FUNCTION_BLOCK "TYPIC_C401_IF_RSS"   // FB106, FBD
TITLE = TYPIC_C401_IF_RSS: RSS-bord
{ S7_Optimized_Access := 'TRUE' }
AUTHOR : OCOTECH
FAMILY : Typical
NAME : C401.701
// Logisch Object Besturing: C401.701
// 
// De interne functie RSSobord verzorgt de bewaking van een RSSobord en stuurt de informatie door naar de subfunctie.
// stored: MemoryReserve 10, SetENOAutomatically false
   VAR_INPUT
      EXT_AUT { ExternalAccessible := 'False'; ExternalVisible := 'False'; ExternalWritable := 'False'} : Bool;   // Externe (hoofd) beveiliging (1 = OK)
      EXT_HW { ExternalAccessible := 'False'; ExternalVisible := 'False'; ExternalWritable := 'False'} : Bool;   // Sturings hardware (PLC) bewaking (1 = OK)
      IN_STO_NOK { ExternalAccessible := 'False'; ExternalVisible := 'False'; ExternalWritable := 'False'} : Bool;   // Storing aanwezig die niet observeerbaar tot gevolg heeft
      IN_STO_OK { ExternalAccessible := 'False'; ExternalVisible := 'False'; ExternalWritable := 'False'} : Bool;   // Storing aanwezig die observeerbaarheid niet beinvloed
      IN_LUS_STO { ExternalAccessible := 'False'; ExternalVisible := 'False'; ExternalWritable := 'False'} : Bool;   // Storing van het luspaar
      IN_STS { ExternalAccessible := 'False'; ExternalVisible := 'False'; ExternalWritable := 'False'} : String[8];   // Naam van de getoonde beeldstand (bitmap) op het bord
      IN_PRTG_STO { ExternalAccessible := 'False'; ExternalVisible := 'False'; ExternalWritable := 'False'} : Bool;   // Storingsmelding RSS-bord vanuit PRTG
      IN_AUT_C401 { ExternalAccessible := 'False'; ExternalVisible := 'False'; ExternalWritable := 'False'} : Bool;   // Beveiligingen: serie geschakelde terugmelding (1 = OK)
   END_VAR
   VAR_OUTPUT
      VAR_IF_RSS { ExternalAccessible := 'False'; ExternalVisible := 'False'; ExternalWritable := 'False'} : "C401_VAR_IF_RSS_TYPIC";   // Struct met alle variabelen naar bovenliggende functies
   END_VAR
   VAR
      STO { ExternalWritable := 'False'} : Struct   // Storingen
         A001 { ExternalAccessible := 'False'; ExternalVisible := 'False'} : Bool;   // Beveiliging aangesproken
         A002 { ExternalAccessible := 'False'; ExternalVisible := 'False'} : Bool;   // Storing luspaar
         A003 { ExternalAccessible := 'False'; ExternalVisible := 'False'} : Bool;   // Storing RSS-bord gedetecteerd door PRTG
         A004 { ExternalAccessible := 'False'; ExternalVisible := 'False'} : Bool;   // Storing RSS-bord
         A005 { ExternalAccessible := 'False'; ExternalVisible := 'False'} : Bool;   // Algemene storing RSS-bord
      END_STRUCT;
      VAR { ExternalWritable := 'False'} : Struct   // Variabelen
         STS { ExternalAccessible := 'False'; ExternalVisible := 'False'} : String[8];   // Naam van de getoonde beeldstand (bitmap) op het bord
         EXT_AUT { ExternalAccessible := 'False'; ExternalVisible := 'False'} : Bool;   // Externe (hoofd) beveiliging aangesproken
         EXT_HW { ExternalAccessible := 'False'; ExternalVisible := 'False'} : Bool;   // Sturings hardware (PLC) in storing
      END_STRUCT;
   END_VAR
BEGIN

REGION Network 1: START
END_REGION

REGION Network 2: +++ Storingen +++
   // Verzamelen storingsmeldingen.
END_REGION

REGION Network 3: Storing A001: Beveiliging aangesproken
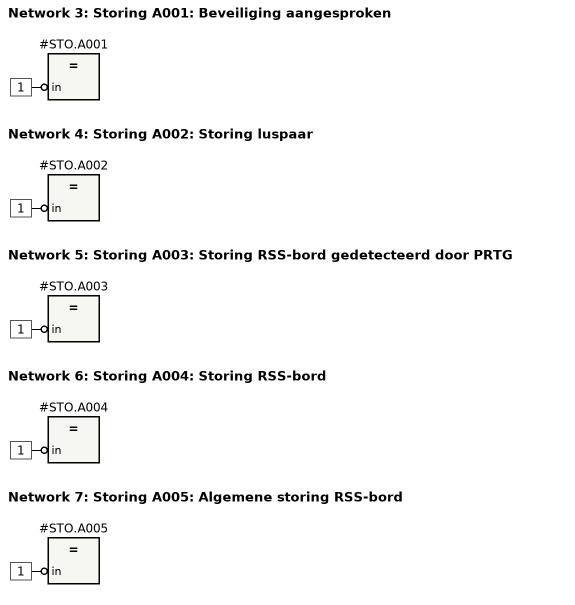
   #STO.A001 := NOT 1;
END_REGION

REGION Network 4: Storing A002: Storing luspaar
   #STO.A002 := NOT 1;
END_REGION

REGION Network 5: Storing A003: Storing RSS-bord gedetecteerd door PRTG
   #STO.A003 := NOT 1;
END_REGION

REGION Network 6: Storing A004: Storing RSS-bord
   #STO.A004 := NOT 1;
END_REGION

REGION Network 7: Storing A005: Algemene storing RSS-bord
   #STO.A005 := NOT 1;
END_REGION

REGION Network 8: +++ Beeldstand +++
   // Doorgeven van de status van het RSS-bord naar de subfunctie.
END_REGION

REGION Network 9 (SCL): EINDE
   // Variabelen van intern scada rakvlak naar outputs copieren
   #VAR_IF_RSS.STS := #VAR.STS;
   #VAR_IF_RSS.EXT_AUT := #VAR.EXT_AUT;
   #VAR_IF_RSS.EXT_HW := #VAR.EXT_HW;
   #VAR_IF_RSS.STO := #STO;
END_REGION
END_FUNCTION_BLOCK

FUNCTION_BLOCK "TYPIC_C402_IF_M33"   // FB110, FBD
TITLE = TYPIC_C402_IF_M33: Voorwaarschuwingsbord
{ S7_Optimized_Access := 'TRUE' }
AUTHOR : OCOTECH
FAMILY : Typical
NAME : C402.703
// Logisch Object Besturing: C402.703
// 
// De interne functie M33 verzorgt de interne besturing van een M33obord.
// 
// Een M33obord is een waarschuwingsbord “verkeerslichten”. Dit bord waarschuwt het verkeer dat zij een actief verkeerslicht naderen.
// 
// Via het DVMosysteem worden de storingsmeldingen van ieder M33obord ingelezen. DVM meldt op zijn beurt storingen van iedere M33obord rechtstreeks aan 3B. De interne besturing heeft geen communicatie met DVM.
// stored: MemoryReserve 10, SetENOAutomatically false
   VAR_INPUT
      EXT_AUT { ExternalAccessible := 'False'; ExternalVisible := 'False'; ExternalWritable := 'False'} : Bool;   // Externe (hoofd) beveiliging (1 = OK)
      EXT_HW { ExternalAccessible := 'False'; ExternalVisible := 'False'; ExternalWritable := 'False'} : Bool;   // Sturings hardware (PLC) bewaking (1 = OK)
      IN_STO_NOK { ExternalAccessible := 'False'; ExternalVisible := 'False'; ExternalWritable := 'False'} : Bool;   // Storing aanwezig die niet observeerbaar tot gevolg heeft
      IN_STO_OK { ExternalAccessible := 'False'; ExternalVisible := 'False'; ExternalWritable := 'False'} : Bool;   // Storing aanwezig die observeerbaarheid niet beinvloed
      IN_PRTG_STO { ExternalAccessible := 'False'; ExternalVisible := 'False'; ExternalWritable := 'False'} : Bool;   // Storingsmelding RSS-bord vanuit PRTG
      IN_AUT_C402 { ExternalAccessible := 'False'; ExternalVisible := 'False'; ExternalWritable := 'False'} : Bool;   // Serie geschakelde beveiligingen (1 = OK)
      IN_AAN { ExternalAccessible := 'False'; ExternalVisible := 'False'; ExternalWritable := 'False'} : Bool;   // Terugmelding aansturing M33-bord (1 = AAN)
      CFG_TYD_FB { ExternalAccessible := 'False'; ExternalVisible := 'False'; ExternalWritable := 'False'} : Time;   // Vertragingstijd storing foute terugmelding
   END_VAR
   VAR_OUTPUT
      VAR_IF_M33 { ExternalAccessible := 'False'; ExternalVisible := 'False'; ExternalWritable := 'False'} : "C402_VAR_IF_M33_TYPIC";   // Struct met alle variabelen naar bovenliggende functies
      OUT_AAN { ExternalAccessible := 'False'; ExternalVisible := 'False'; ExternalWritable := 'False'} : Bool;   // Aansturing M33-bord (TRUE = Uit / FALSE = Aan)
   END_VAR
   VAR_IN_OUT
      STU_IF_M33 : "C402_STU_IF_M33_TYPIC";   // Struct met alle sturingen van de subfunctie (SF) M33 van 3B
   END_VAR
   VAR
      STO { ExternalWritable := 'False'} : Struct   // Storingen
         A001 { ExternalAccessible := 'False'; ExternalVisible := 'False'} : Bool;   // Beveiliging aangesproken
         A002 { ExternalAccessible := 'False'; ExternalVisible := 'False'} : Bool;   // Storing M33-bord gedetecteerd door PRTG
         A003 { ExternalAccessible := 'False'; ExternalVisible := 'False'} : Bool;   // Storing M33-bord
         A004 { ExternalAccessible := 'False'; ExternalVisible := 'False'} : Bool;   // Algemene storing M33-bord
         AT01 { ExternalAccessible := 'False'; ExternalVisible := 'False'} : Bool;   // Foute terugmelding: M33-bord aangestuurd, terugmelding Aan niet (of te laat) ontvangen
         AT02 { ExternalAccessible := 'False'; ExternalVisible := 'False'} : Bool;   // Foute terugmelding: M33-bord niet aangestuurd, terugmelding Aan blijft aanwezig
      END_STRUCT;
      VAR { ExternalWritable := 'False'} : Struct   // Variabelen
         STS_AAN { ExternalAccessible := 'False'; ExternalVisible := 'False'} : Bool;   // TRUE = M33-bord actueel in werking FALSE = Uit
         EXT_AUT { ExternalAccessible := 'False'; ExternalVisible := 'False'} : Bool;   // Externe (hoofd) beveiliging aangesproken
         EXT_HW { ExternalAccessible := 'False'; ExternalVisible := 'False'} : Bool;   // Sturings hardware (PLC) in storing
      END_STRUCT;
   END_VAR
BEGIN

REGION Network 1: START
END_REGION

REGION Network 2: +++ Aansturing bord +++
   // Aansturen bord en terugmeldingsbewaking (Aan / Uit).
END_REGION

REGION Network 3: +++ Storingen +++
   // Verwerken van de storingsmeldingen.
END_REGION

REGION Network 4: Storing A001: Beveiliging aangesproken
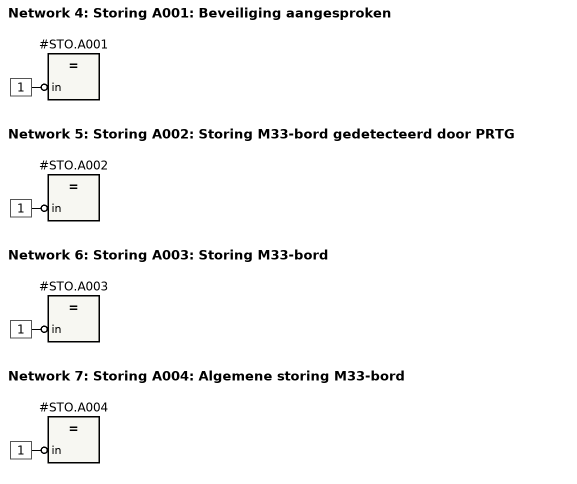
   #STO.A001 := NOT 1;
END_REGION

REGION Network 5: Storing A002: Storing M33-bord gedetecteerd door PRTG
   #STO.A002 := NOT 1;
END_REGION

REGION Network 6: Storing A003: Storing M33-bord
   #STO.A003 := NOT 1;
END_REGION

REGION Network 7: Storing A004: Algemene storing M33-bord
   #STO.A004 := NOT 1;
END_REGION

REGION Network 8 (SCL): EINDE
   // Variabelen van intern scada rakvlak naar outputs copieren
   #VAR_IF_M33.STS_AAN := #VAR.STS_AAN;
   #VAR_IF_M33.EXT_AUT := #VAR.EXT_AUT;
   #VAR_IF_M33.EXT_HW := #VAR.EXT_HW;
   #VAR_IF_M33.STO := #STO;
END_REGION
END_FUNCTION_BLOCK

FUNCTION_BLOCK "TYPIC_C402_IF_SBO1"   // FB111, FBD
TITLE = TYPIC_C402_IF_SBO: Afsluitboom
{ S7_Optimized_Access := 'TRUE' }
AUTHOR : OCOTECH
FAMILY : Typical
NAME : C402.704
// Logisch Object Besturing: C402.704
// 
// 								De interne functie afsluitboom verzorgt de interne besturing,
// 								bewaking en fysieke aansturing van een afsluitboom.
// 
// 								Het akoestisch signaal en de optische signalen behorend bij de
// 								afsluitboom, wordt eveneens via deze functie aangestuurd.
// stored: MemoryReserve 10, SetENOAutomatically false
   VAR_INPUT
      EXT_AUT { ExternalAccessible := 'False'; ExternalVisible := 'False'; ExternalWritable := 'False'} : Bool;   // Externe (hoofd) beveiliging (1 = OK)
      EXT_HW { ExternalAccessible := 'False'; ExternalVisible := 'False'; ExternalWritable := 'False'} : Bool;   // Sturings hardware (PLC) bewaking (1 = OK)
      HULP_KNIP { ExternalAccessible := 'False'; ExternalVisible := 'False'; ExternalWritable := 'False'} : Bool;   // Knippersignaal, x tijd hoog, x tijd laag
      IN_AUT { ExternalAccessible := 'False'; ExternalVisible := 'False'; ExternalWritable := 'False'} : Bool;   // Motorbeveiliging (1 = OK / 0 = storing)
      IN_OPEN { ExternalAccessible := 'False'; ExternalVisible := 'False'; ExternalWritable := 'False'} : Bool;   // Terugmelding: afsluitboom is open
      IN_TOE { ExternalAccessible := 'False'; ExternalVisible := 'False'; ExternalWritable := 'False'} : Bool;   // Terugmelding: afsluitboom is toe
      IN_STO { ExternalAccessible := 'False'; ExternalVisible := 'False'; ExternalWritable := 'False'} : Bool;   // Terugmelding: afsluitboom is buiten dienst
      IN_SCW { ExternalAccessible := 'False'; ExternalVisible := 'False'; ExternalWritable := 'False'} : Bool;   // Werkschakelaar (1 = AAN)
      IN_HND { ExternalAccessible := 'False'; ExternalVisible := 'False'; ExternalWritable := 'False'} : Bool;   // Mechanische handmatige bediening (0 = Hand)
      IN_LVE1_STO { ExternalAccessible := 'False'; ExternalVisible := 'False'; ExternalWritable := 'False'} : Bool;   // Detector lus 1 (1 = OK / 0 = storing)
      IN_LVE2_STO { ExternalAccessible := 'False'; ExternalVisible := 'False'; ExternalWritable := 'False'} : Bool;   // Detector lus 2 (1 = OK / 0 = storing)
      IN_LVE3_STO { ExternalAccessible := 'False'; ExternalVisible := 'False'; ExternalWritable := 'False'} : Bool;   // Detector lus 3 (1 = OK / 0 = storing)
      IN_LVE4_STO { ExternalAccessible := 'False'; ExternalVisible := 'False'; ExternalWritable := 'False'} : Bool;   // Detector lus 4 (1 = OK / 0 = storing)
      IN_LUS1_STS { ExternalAccessible := 'False'; ExternalVisible := 'False'; ExternalWritable := 'False'} : Bool;   // Detectie voertuig door lus 1 (1 = Geen detectie)
      IN_LUS2_STS { ExternalAccessible := 'False'; ExternalVisible := 'False'; ExternalWritable := 'False'} : Bool;   // Detectie voertuig door lus 2 (1 = Geen detectie)
      IN_LUS3_STS { ExternalAccessible := 'False'; ExternalVisible := 'False'; ExternalWritable := 'False'} : Bool;   // Detectie voertuig door lus 3 (1 = Geen detectie)
      IN_LUS4_STS { ExternalAccessible := 'False'; ExternalVisible := 'False'; ExternalWritable := 'False'} : Bool;   // Detectie voertuig door lus 4 (1 = Geen detectie)
      IN_AUT_C402 { ExternalAccessible := 'False'; ExternalVisible := 'False'; ExternalWritable := 'False'} : Bool;   // Beveiligingen: serie geschakelde terugmelding (1 = OK)
      IN_DKN_OPEN { ExternalAccessible := 'False'; ExternalVisible := 'False'; ExternalWritable := 'False'} : Bool;   // 1 = Drukknop ingedrukt, bediening openen
      IN_DKN_TOE { ExternalAccessible := 'False'; ExternalVisible := 'False'; ExternalWritable := 'False'} : Bool;   // 1 = Drukknop ingedrukt, bediening sluiten
      IN_DKN_STOP { ExternalAccessible := 'False'; ExternalVisible := 'False'; ExternalWritable := 'False'} : Bool;   // 1 = Drukknop ingedrukt, bediening stop
      CFG_TYD_STS { ExternalAccessible := 'False'; ExternalVisible := 'False'; ExternalWritable := 'False'} : Time;   // Vertragingstijd storing terugmelding stand bereikt
      CFG_ITYD_POS { ExternalAccessible := 'False'; ExternalVisible := 'False'; ExternalWritable := 'False'} : Time;   // Inschakelvertraging storing eindpositie terugmelding weggevallen
      CFG_UTYD_POS { ExternalAccessible := 'False'; ExternalVisible := 'False'; ExternalWritable := 'False'} : Time;   // Uitschakelvertraging storing eindpositie terugmelding weggevallen
      CFG_ITYD_OAS_SNEL { ExternalAccessible := 'False'; ExternalVisible := 'False'; ExternalWritable := 'False'} : Time;   // Vertragingstijd versneld sluiten afsluitboom na akoestisch en optisch signaal
      CFG_ITYD_OAS { ExternalAccessible := 'False'; ExternalVisible := 'False'; ExternalWritable := 'False'} : Time;   // Vertragingstijd sluiten/openen afsluitboom regulier na akoestisch en optisch signaal
      CFG_UTYD_OAS { ExternalAccessible := 'False'; ExternalVisible := 'False'; ExternalWritable := 'False'} : Time;   // Vertragingstijd uitschakelen akoestische en optische signalen
      CFG_UTYD_MOT { ExternalAccessible := 'False'; ExternalVisible := 'False'; ExternalWritable := 'False'} : Time;   // Vertragingstijd uitschakelen motor na bereiken eindpositie
      CFG_VGV_OPEN { ExternalAccessible := 'False'; ExternalVisible := 'False'; ExternalWritable := 'False'} : Bool;   // 1 = Slagboom moet openen bij bediening openen door hulpdiensten
   END_VAR
   VAR_OUTPUT
      VAR_IF_SBO { ExternalAccessible := 'False'; ExternalVisible := 'False'; ExternalWritable := 'False'} : "C402_VAR_IF_SBO_TYPIC";   // Struct met alle variabelen naar bovenliggende functies
      OUT_OPEN { ExternalAccessible := 'False'; ExternalVisible := 'False'; ExternalWritable := 'False'} : Bool;   // Aansturing openen
      OUT_TOE { ExternalAccessible := 'False'; ExternalVisible := 'False'; ExternalWritable := 'False'} : Bool;   // Aansturing sluiten
      OUT_AKS { ExternalAccessible := 'False'; ExternalVisible := 'False'; ExternalWritable := 'False'} : Bool;   // Aansturen akoestische signalering
      OUT_OPS { ExternalAccessible := 'False'; ExternalVisible := 'False'; ExternalWritable := 'False'} : Bool;   // Aansturen optische signalering
   END_VAR
   VAR_IN_OUT
      STU_IF_SBO : "C402_STU_IF_SBO_TYPIC";   // Struct met alle sturingen naar de functie (IF) in de interne sturing van de afsluitboom
      STU_AFS_IF_SBO : "C402_STU_AFS_IF_SBO_TYPIC";   // Struct met alle sturingen vanuit de interne functie Afsluitsysteem naar de functies (IF) van de afsluitbomen
   END_VAR
   VAR
      STO { ExternalWritable := 'False'} : Struct   // Storingen
         A001 { ExternalAccessible := 'False'; ExternalVisible := 'False'} : Bool;   // Beveiliging aangesproken
         A002 { ExternalAccessible := 'False'; ExternalVisible := 'False'} : Bool;   // Storing van de detector van lus 1
         A003 { ExternalAccessible := 'False'; ExternalVisible := 'False'} : Bool;   // Storing van de detector van lus 2
         A004 { ExternalAccessible := 'False'; ExternalVisible := 'False'} : Bool;   // Storing van de detector van lus 3
         A005 { ExternalAccessible := 'False'; ExternalVisible := 'False'} : Bool;   // Storing van de detector van lus 4
         A006 { ExternalAccessible := 'False'; ExternalVisible := 'False'} : Bool;   // Storing van de motorsturing
         A007 { ExternalAccessible := 'False'; ExternalVisible := 'False'} : Bool;   // Storing motorbeveiliging
         AT01 { ExternalAccessible := 'False'; ExternalVisible := 'False'} : Bool;   // Terugmelding Open niet tijdig bereikt
         AT02 { ExternalAccessible := 'False'; ExternalVisible := 'False'} : Bool;   // Terugmelding Dicht niet tijdig bereikt
         AT03 { ExternalAccessible := 'False'; ExternalVisible := 'False'} : Bool;   // Terugmeldingen Open en Dicht tegelijkertijd
         AT04 { ExternalAccessible := 'False'; ExternalVisible := 'False'} : Bool;   // Terugmelding Open weggevallen
         AT05 { ExternalAccessible := 'False'; ExternalVisible := 'False'} : Bool;   // Terugmelding Dicht weggevallen
         M001 { ExternalAccessible := 'False'; ExternalVisible := 'False'} : Bool;   // Werkschakelaar uitgeschakeld
         M002 { ExternalAccessible := 'False'; ExternalVisible := 'False'} : Bool;   // Mechanische handbediening uitgenomen
      END_STRUCT;
      VAR { ExternalWritable := 'False'} : Struct   // Variabelen
         CMD_AKS { ExternalAccessible := 'False'; ExternalVisible := 'False'} : Bool;   // Aansturen akoestische signalering
         CMD_OPS { ExternalAccessible := 'False'; ExternalVisible := 'False'} : Bool;   // Aansturen optische signalering
         VWA_AT04 { ExternalAccessible := 'False'; ExternalVisible := 'False'} : Bool;   // Voorwaarden voldaan voor storing AT04
         VWA_AT05 { ExternalAccessible := 'False'; ExternalVisible := 'False'} : Bool;   // Voorwaarden voldaan voor storing AT05
         MOT_STS_AAN { ExternalAccessible := 'False'; ExternalVisible := 'False'} : Bool;   // Motor afsluitboom aangestuurd
         CMD_OPEN { ExternalAccessible := 'False'; ExternalVisible := 'False'} : Bool;   // Gewenste stand afsluitboom is Open
         CMD_TOE { ExternalAccessible := 'False'; ExternalVisible := 'False'} : Bool;   // Gewenste stand afsluitboom is Toe
         CMD_STOP { ExternalAccessible := 'False'; ExternalVisible := 'False'} : Bool;   // Gewenste stand afsluitboom is Stop
         STO { ExternalAccessible := 'False'; ExternalVisible := 'False'} : Bool;   // De afsluitboom heeft een storing waardoor deze niet aangestuurd kan worden
         LOK_OPEN { ExternalAccessible := 'False'; ExternalVisible := 'False'} : Bool;   // Afsluitboom dient te openen voor hulpdiensten
         CMD_NEW { ExternalAccessible := 'False'; ExternalVisible := 'False'} : Bool;   // Nieuwe commando ontvangen vanuit 3B
         VGV_TOE { ExternalAccessible := 'False'; ExternalVisible := 'False'} : Bool;   // Vrijgave om de afsluitboom te sluiten
         CMD_TYD_OPEN { ExternalAccessible := 'False'; ExternalVisible := 'False'} : Bool;   // Gewenste stand afsluitboom is Open, tijdsvertraging OK
         CMD_TYD_TOE { ExternalAccessible := 'False'; ExternalVisible := 'False'} : Bool;   // Gewenste stand afsluitboom is Toe, tijdsvertraging OK
         STS_BEZ_OPEN { ExternalAccessible := 'False'; ExternalVisible := 'False'} : Bool;   // TRUE = Afsluitboom bezig met beweging openen
         STS_BEZ_TOE { ExternalAccessible := 'False'; ExternalVisible := 'False'} : Bool;   // TRUE = Afsluitboom bezig met beweging sluiten
         STS_OPEN { ExternalAccessible := 'False'; ExternalVisible := 'False'} : Bool;   // TRUE = Afsluitboom op stand Open
         STS_TOE { ExternalAccessible := 'False'; ExternalVisible := 'False'} : Bool;   // TRUE = Afsluitboom op stand Dicht
         STS_STOP { ExternalAccessible := 'False'; ExternalVisible := 'False'} : Bool;   // TRUE = Afsluitboom niet op een eindpositie en niet in beweging
         BMO_HAND { ExternalAccessible := 'False'; ExternalVisible := 'False'} : Bool;   // TRUE = Afsluitboom in hand geschakeld / FALSE = niet in hand
         STS_VKL_OK { ExternalAccessible := 'False'; ExternalVisible := 'False'} : Bool;   // TRUE = Verkeerslichten op Rood (voorwaarde voor sluiten)
         STS_NDS_OK { ExternalAccessible := 'False'; ExternalVisible := 'False'} : Bool;   // TRUE = Geen noodstop (voorwaarde voor beweging)
         STS_LUS_OK { ExternalAccessible := 'False'; ExternalVisible := 'False'} : Bool;   // TRUE = Detectielus(sen) OK (geen obstakel gedetecteerd voor sluiten)
         EXT_AUT { ExternalAccessible := 'False'; ExternalVisible := 'False'} : Bool;   // Externe (hoofd) beveiliging aangesproken
         EXT_HW { ExternalAccessible := 'False'; ExternalVisible := 'False'} : Bool;   // Sturings hardware (PLC) in storing
         EXT_STO { ExternalAccessible := 'False'; ExternalVisible := 'False'} : Bool;   // Externe storing aanwezig
         LUS1_STS { ExternalAccessible := 'False'; ExternalVisible := 'False'} : Bool;   // Detectie voertuig door lus 1 (1 = detectie)
         LUS2_STS { ExternalAccessible := 'False'; ExternalVisible := 'False'} : Bool;   // Detectie voertuig door lus 2 (1 = detectie)
         LUS3_STS { ExternalAccessible := 'False'; ExternalVisible := 'False'} : Bool;   // Detectie voertuig door lus 3 (1 = detectie)
         LUS4_STS { ExternalAccessible := 'False'; ExternalVisible := 'False'} : Bool;   // Detectie voertuig door lus 3 (1 = detectie)
      END_STRUCT;
   END_VAR
BEGIN

REGION Network 1: START
END_REGION

REGION Network 2: +++ Storingen en meldingen +++
   // Verwerken van de storingen en meldingen.
END_REGION

REGION Network 3: Storing A001: Beveiliging aangesproken
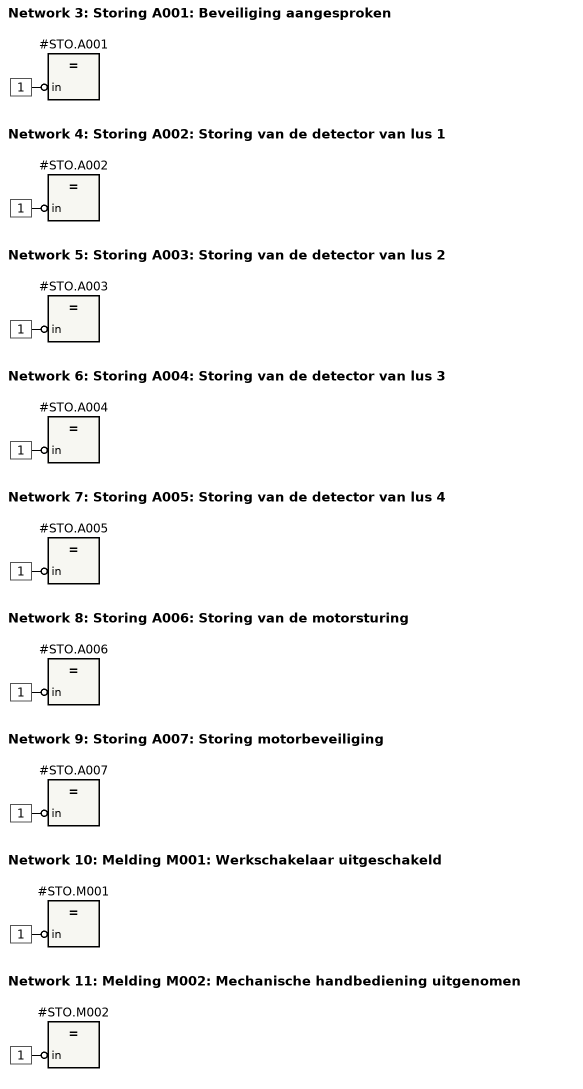
   #STO.A001 := NOT 1;
END_REGION

REGION Network 4: Storing A002: Storing van de detector van lus 1
   #STO.A002 := NOT 1;
END_REGION

REGION Network 5: Storing A003: Storing van de detector van lus 2
   #STO.A003 := NOT 1;
END_REGION

REGION Network 6: Storing A004: Storing van de detector van lus 3
   #STO.A004 := NOT 1;
END_REGION

REGION Network 7: Storing A005: Storing van de detector van lus 4
   #STO.A005 := NOT 1;
END_REGION

REGION Network 8: Storing A006: Storing van de motorsturing
   #STO.A006 := NOT 1;
END_REGION

REGION Network 9: Storing A007: Storing motorbeveiliging
   #STO.A007 := NOT 1;
END_REGION

REGION Network 10: Melding M001: Werkschakelaar uitgeschakeld
   #STO.M001 := NOT 1;
END_REGION

REGION Network 11: Melding M002: Mechanische handbediening uitgenomen
   #STO.M002 := NOT 1;
END_REGION

REGION Network 12: +++ Status detectielussen +++
   // De afsluitboom kan enkel voorwaardelijk sluiten als de
   // 										detectielussen geen metalen object detecteren en geen
   // 										storing hebben.
END_REGION

REGION Network 13: +++ Openen afsluitboom voor hulpdiensten +++
   // De afsluitboom kan door de hulpdiensten geopend worden als
   // 										op het bedieningspaneel de betreffende drukknop bediend
   // 										wordt en er vrijgave is voor bediening.
END_REGION

REGION Network 14: +++ Gewenste beweging afsluitboom +++
   // Afhankelijk van de werkingsmode, bedieningen en commandos
   // 										wordt de gewenste beweging van de afsluitboom bepaald
   // 										(openen / sluiten / stop).
END_REGION

REGION Network 15: +++ Vrijgave sluiten +++
   // Het sluiten van de afsluitboom mag enkel plaatsvinden als
   // 										er geen obstakel gedetecteerd wordt. Bij handbediening of
   // 										bij het commando onvoorwaardelijk sluiten wordt er geen
   // 										rekening gehouden met de obstakeldetectie.
END_REGION

REGION Network 16: +++ Tijdsvertraging aansturen afsluitboom +++
   // Vooraleer de afsluitboom aan te sturen, dienen de
   // 										akoestische en optische signalering aangestuurd te zijn. Pas
   // 										na een korte tijdsvertraging mag de afsluitboom in beweging
   // 										komen.
END_REGION

REGION Network 17: +++ Afsluitboomsturing +++
   // Aansturen van de afsluitboom en terugmeldingsbewaking.
END_REGION

REGION Network 18: +++ Sturing akoestische signalering +++
   // De akoestische signalering wordt aangestuurd van zodra de
   // 										afsluitboom dient te bewegen. De beweging wordt pas ingezet
   // 										nadat de akoestische signalering gedurende een bepaalde tijd
   // 										aangestuurd geweest is.
END_REGION

REGION Network 19: +++ Sturing Optische signalering +++
   // De optische signalering wordt aangestuurd van zodra de
   // 										afsluitboom dient te bewegen en blijft aangestuurd tot de
   // 										afsluitboom zich opnieuw in de open positie bevindt.
END_REGION

REGION Network 20 (SCL): EINDE
   // Variabelen van intern scada rakvlak naar outputs copieren
   #VAR_IF_SBO.STS_BEZ_OPEN := #VAR.STS_BEZ_OPEN;
   #VAR_IF_SBO.STS_BEZ_TOE := #VAR.STS_BEZ_TOE;
   #VAR_IF_SBO.STS_OPEN := #VAR.STS_OPEN;
   #VAR_IF_SBO.STS_TOE := #VAR.STS_TOE;
   #VAR_IF_SBO.STS_STOP := #VAR.STS_STOP;
   #VAR_IF_SBO.BMO_HAND := #VAR.BMO_HAND;
   #VAR_IF_SBO.STS_VKL_OK := #VAR.STS_VKL_OK;
   #VAR_IF_SBO.STS_NDS_OK := #VAR.STS_NDS_OK;
   #VAR_IF_SBO.STS_LUS_OK := #VAR.STS_LUS_OK;
   #VAR_IF_SBO.EXT_AUT := #VAR.EXT_AUT;
   #VAR_IF_SBO.EXT_HW := #VAR.EXT_HW;
   #VAR_IF_SBO.EXT_STO := #VAR.EXT_STO;
   #VAR_IF_SBO.LUS1_STS := #VAR.LUS1_STS;
   #VAR_IF_SBO.LUS2_STS := #VAR.LUS2_STS;
   #VAR_IF_SBO.LUS3_STS := #VAR.LUS3_STS;
   #VAR_IF_SBO.LUS4_STS := #VAR.LUS4_STS;
   #VAR_IF_SBO.STO := #STO;
END_REGION
END_FUNCTION_BLOCK

FUNCTION_BLOCK "TYPIC_C402_IF_VKL"   // FB112, FBD
TITLE = TYPIC_C402_IF_VKL: Verkeerslicht
{ S7_Optimized_Access := 'TRUE' }
AUTHOR : OCOTECH
FAMILY : Typical
NAME : C402.702
// Logisch Object Besturing: C402.702
// 
// De interne functie verkeerslicht verzorgt de interne besturing, bewaking en fysieke aansturing van een verkeerslicht.
// 
// Het verkeerslicht kan via sturingen (vanuit 3B) of via handmatige bedieningen (aanraakscherm) op volgende standen gezet worden:
//  UIT (gedoofd)
//  ROOD
//  GROEN
//  GEEL KNIPPEREN
// 
// De stand “Geel vast” kan niet via sturing of bediening gekozen worden. De stand “Geel vast” wordt door deze typical altijd automatisch toegepast als overgang naar stand “Rood”.
// stored: MemoryReserve 10, SetENOAutomatically false
   VAR_INPUT
      EXT_AUT { ExternalAccessible := 'False'; ExternalVisible := 'False'; ExternalWritable := 'False'} : Bool;   // Externe (hoofd) beveiliging (1 = OK)
      EXT_HW { ExternalAccessible := 'False'; ExternalVisible := 'False'; ExternalWritable := 'False'} : Bool;   // Sturings hardware (PLC) bewaking (1 = OK)
      HULP_KNIP { ExternalAccessible := 'False'; ExternalVisible := 'False'; ExternalWritable := 'False'} : Bool;   // Knippersignaal, x tijd Hoog, x tijd Laag
      IN_AUT_C402 { ExternalAccessible := 'False'; ExternalVisible := 'False'; ExternalWritable := 'False'} : Bool;   // Beveiligingen: serie geschakelde terugmelding (1 = OK)
      IN_ROOD { ExternalAccessible := 'False'; ExternalVisible := 'False'; ExternalWritable := 'False'} : Bool;   // Terugmelding: rood aan (stroommeting)
      IN_GEEL { ExternalAccessible := 'False'; ExternalVisible := 'False'; ExternalWritable := 'False'} : Bool;   // Terugmelding: geel aan (stroommeting)
      IN_GROE { ExternalAccessible := 'False'; ExternalVisible := 'False'; ExternalWritable := 'False'} : Bool;   // Terugmelding: groen aan (stroommeting)
      CFG_TYD_FB { ExternalAccessible := 'False'; ExternalVisible := 'False'; ExternalWritable := 'False'} : Time;   // Vertragingstijd storing terugmelding
      CFG_GEEL_TYD { ExternalAccessible := 'False'; ExternalVisible := 'False'; ExternalWritable := 'False'} : Time;   // Tijdsduur verkeerslicht geel, vooraleer naar rood
      CFG_SNEL_GEEL_TYD { ExternalAccessible := 'False'; ExternalVisible := 'False'; ExternalWritable := 'False'} : Time;   // Tijdsduur verkeerslicht geel, vooraleer naar rood, bij versneld sluiten
      CFG_TYD_ONHD { ExternalAccessible := 'False'; ExternalVisible := 'False'; ExternalWritable := 'False'} : Time;   // Tijdsduur aansturing lenzen bij automatische onderhoudstesten
   END_VAR
   VAR_OUTPUT
      VAR_IF_VKL { ExternalAccessible := 'False'; ExternalVisible := 'False'; ExternalWritable := 'False'} : "C402_VAR_IF_VKL_TYPIC";   // Struct met alle variabelen naar bovenliggende functies
      OUT_ROOD { ExternalAccessible := 'False'; ExternalVisible := 'False'; ExternalWritable := 'False'} : Bool;   // Aansturing rood
      OUT_GEEL { ExternalAccessible := 'False'; ExternalVisible := 'False'; ExternalWritable := 'False'} : Bool;   // Aansturing geel
      OUT_GROE { ExternalAccessible := 'False'; ExternalVisible := 'False'; ExternalWritable := 'False'} : Bool;   // Aansturing groen
   END_VAR
   VAR_IN_OUT
      STU_IF_VKL : "C402_STU_IF_VKL_TYPIC";   // Struct met alle sturingen naar de functie (IF) in de interne sturing van het verkeerslicht
      STU_AFS_IF_VKL : "C402_STU_AFS_IF_VKL_TYPIC";   // Struct met alle sturingen naar de functie (IF) van de verkeerslichten
   END_VAR
   VAR
      STO { ExternalWritable := 'False'} : Struct   // Storingen
         A001 { ExternalAccessible := 'False'; ExternalVisible := 'False'} : Bool;   // Beveiliging aangesproken
         AT01 { ExternalAccessible := 'False'; ExternalVisible := 'False'} : Bool;   // De rode lens is defect
         AT02 { ExternalAccessible := 'False'; ExternalVisible := 'False'} : Bool;   // De gele lens is defect
         AT03 { ExternalAccessible := 'False'; ExternalVisible := 'False'} : Bool;   // De groene lens is defect
         AT04 { ExternalAccessible := 'False'; ExternalVisible := 'False'} : Bool;   // De stand rood kan niet getoond worden
         AT05 { ExternalAccessible := 'False'; ExternalVisible := 'False'} : Bool;   // De stand geel kan niet getoond worden
         AT06 { ExternalAccessible := 'False'; ExternalVisible := 'False'} : Bool;   // De stand geel knipperen kan niet getoond worden
         AT07 { ExternalAccessible := 'False'; ExternalVisible := 'False'} : Bool;   // De stand groen kan niet getoond worden
      END_STRUCT;
      VAR { ExternalWritable := 'False'} : Struct   // Variabelen
         HAND_ROOD_SWA { ExternalAccessible := 'False'; ExternalVisible := 'False'} : Bool;   // 1 = Rood gewenst, via handbediening
         HAND_KNIP_SWA { ExternalAccessible := 'False'; ExternalVisible := 'False'} : Bool;   // 1 = Geel knipperen gewenst, via handbediening
         HAND_GROE_SWA { ExternalAccessible := 'False'; ExternalVisible := 'False'} : Bool;   // 1 = Groen gewenst, via handbediening
         ROOD_SWA { ExternalAccessible := 'False'; ExternalVisible := 'False'} : Bool;   // 1 = Rood gewenst
         KNIP_SWA { ExternalAccessible := 'False'; ExternalVisible := 'False'} : Bool;   // 1 = Geel knipperen gewenst
         GROEN_SWA { ExternalAccessible := 'False'; ExternalVisible := 'False'} : Bool;   // 1 = Groen gewenst
         ROOD_AAN_SWA { ExternalAccessible := 'False'; ExternalVisible := 'False'} : Bool;   // 1 = Rood gewenst, rode lens aansturen
         GEEL_AAN_SWA { ExternalAccessible := 'False'; ExternalVisible := 'False'} : Bool;   // 1 = Rood gewenst, gele lens aansturen
         GEEL_KNIP { ExternalAccessible := 'False'; ExternalVisible := 'False'} : Bool;   // Knippersignaal voor geel licht 1 = AAN / 0 = UIT
         STO_ROOD_AAN { ExternalAccessible := 'False'; ExternalVisible := 'False'} : Bool;   // 1 = Rode lens defect, geen terugmelding bij aansturen
         STO_ROOD_UIT { ExternalAccessible := 'False'; ExternalVisible := 'False'} : Bool;   // 1 = Rode lens defect, terugmelding aan bij afsturen
         STO_GEEL_AAN { ExternalAccessible := 'False'; ExternalVisible := 'False'} : Bool;   // 1 = Gele lens defect, geen terugmelding bij aansturen
         STO_GEEL_UIT { ExternalAccessible := 'False'; ExternalVisible := 'False'} : Bool;   // 1 = Gele lens defect, terugmelding aan bij afsturen
         STO_GROE_AAN { ExternalAccessible := 'False'; ExternalVisible := 'False'} : Bool;   // 1 = Groene lens defect, geen terugmelding bij aansturen
         STO_GROE_UIT { ExternalAccessible := 'False'; ExternalVisible := 'False'} : Bool;   // 1 = Groene lens defect, terugmelding aan bij afsturen
         ONHD { ExternalAccessible := 'False'; ExternalVisible := 'False'} : Bool;   // 1 = Alle lenzen aansturen ifv onderhoudstesten
         STS_ROOD { ExternalAccessible := 'False'; ExternalVisible := 'False'} : Bool;   // TRUE = Verkeerslicht actueel op rood
         STS_GEEL { ExternalAccessible := 'False'; ExternalVisible := 'False'} : Bool;   // TRUE = Verkeerslicht actueel op geel (vast)
         STS_GROE { ExternalAccessible := 'False'; ExternalVisible := 'False'} : Bool;   // TRUE = Verkeerslicht actueel op groen
         STS_KNIP { ExternalAccessible := 'False'; ExternalVisible := 'False'} : Bool;   // TRUE = Verkeerslicht actueel op knipperen geel
         STS_AAN { ExternalAccessible := 'False'; ExternalVisible := 'False'} : Bool;   // TRUE = Verkeerslicht wordt aangestuurd
         BMO_HAND { ExternalAccessible := 'False'; ExternalVisible := 'False'} : Bool;   // TRUE = Verkeerslicht in hand geschakeld / FALSE = niet in hand
         EXT_AUT { ExternalAccessible := 'False'; ExternalVisible := 'False'} : Bool;   // Externe (hoofd) beveiliging aangesproken
         EXT_HW { ExternalAccessible := 'False'; ExternalVisible := 'False'} : Bool;   // Sturings hardware (PLC) in storing
      END_STRUCT;
   END_VAR
BEGIN

REGION Network 1: START
END_REGION

REGION Network 2: +++ Bepalen bedieningsmode +++
   // Bedieningsmode (Afstand / Hand) bepalen.
END_REGION

REGION Network 3: +++ Bepalen gewenste status +++
   // Gewenste status van het verkeerslicht bepalen (Rood / Geel Knipperen / Groen / Uit).
END_REGION

REGION Network 4: +++ Overgang naar rood +++
   // Als de gewenste stand Rood is, zal er eerst een overgang zijn waarbij het verkeerslicht op geel wordt aangestuurd.
END_REGION

REGION Network 5: +++ Storingen +++
   // Terugmeldingsbewaking van iedere lens.
END_REGION

REGION Network 6: Storing A001: Beveiliging aangesproken
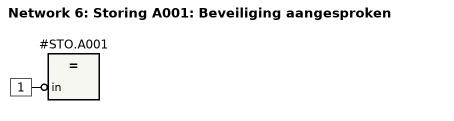
   #STO.A001 := NOT 1;
END_REGION

REGION Network 7: +++ Bepalen actuele status +++
   // Actuele status van het verkeerslicht (Rood / Geel / Geel Knipperen / Groen / Uit).
END_REGION

REGION Network 8: +++ Automatische onderhoudstesten +++
   // Alle lenzen kortstondig en gelijktijdig aansturen ter controle van de goede werking.
END_REGION

REGION Network 9: +++ Aansturing lenzen +++
   // Aansturen van iedere lens (Aan / Uit).
END_REGION

REGION Network 10 (SCL): EINDE
   // Variabelen van intern scada rakvlak naar outputs copieren
   #VAR_IF_VKL.STS_ROOD := #VAR.STS_ROOD;
   #VAR_IF_VKL.STS_GEEL := #VAR.STS_GEEL;
   #VAR_IF_VKL.STS_GROE := #VAR.STS_GROE;
   #VAR_IF_VKL.STS_KNIP := #VAR.STS_KNIP;
   #VAR_IF_VKL.STS_AAN := #VAR.STS_AAN;
   #VAR_IF_VKL.BMO_HAND := #VAR.BMO_HAND;
   #VAR_IF_VKL.EXT_AUT := #VAR.EXT_AUT;
   #VAR_IF_VKL.EXT_HW := #VAR.EXT_HW;
   #VAR_IF_VKL.STO := #STO;
END_REGION
END_FUNCTION_BLOCK

FUNCTION_BLOCK "TYPIC_C403_IF_LVE"   // FB132, FBD
TITLE = TYPIC_C403_IF_LVE: Detectiepunt
{ S7_Optimized_Access := 'TRUE' }
AUTHOR : OCOTECH
FAMILY : Typical
NAME : C403.702
// Logisch Object Besturing: C403.701
// 
// Het doel van de IF LVE (Detectiepunt SnelheidsOnderschrijding) is om de gegevens te verwerken die ontvangen worden van een detectiepunt uit de interne sturing en via inputs.
// stored: MemoryReserve 10, SetENOAutomatically false
   VAR_INPUT
      EXT_HW { ExternalAccessible := 'False'; ExternalVisible := 'False'; ExternalWritable := 'False'} : Bool;   // Sturings hardware (PLC) bewaking (1 = OK)
      IN_AUT_C403 { ExternalAccessible := 'False'; ExternalVisible := 'False'; ExternalWritable := 'False'} : Bool;   // Beveiligingen: serie geschakelde terugmelding (1= OK)
      IN_AUT { ExternalAccessible := 'False'; ExternalVisible := 'False'; ExternalWritable := 'False'} : Bool;   // Beveiliging kastklimatisatie (1 = OK)
      IN_SPD_OK { ExternalAccessible := 'False'; ExternalVisible := 'False'; ExternalWritable := 'False'} : Bool;   // Status overspanningsbeveiliging (1 = OK)
      IN_DEC { ExternalAccessible := 'False'; ExternalVisible := 'False'; ExternalWritable := 'False'} : Bool;   // Deurcontact (1 = Gesloten)
      IN_STS { ExternalAccessible := 'False'; ExternalVisible := 'False'; ExternalWritable := 'False'} : Word;   // Statusbits van een lusdetectie
   END_VAR
   VAR_OUTPUT
      VAR_IF_LVE { ExternalAccessible := 'False'; ExternalVisible := 'False'; ExternalWritable := 'False'} : "C403_VAR_IF_LVE_TYPIC";   // Struct met alle variabelen naar de subfunctie
   END_VAR
   VAR
      STO { ExternalWritable := 'False'} : Struct   // Storingen
         A001 : Bool;   // Beveiliging aangesproken
         A002 : Bool;   // Storing detectiepunt
         A003 : Bool;   // Beveiliging klimaatregeling wegkantkast aangesproken
         A004 : Bool;   // Overspanningsbeveiliging aangesproken
      END_STRUCT;
      VAR { ExternalWritable := 'False'} : Struct   // Variabelen
         EXT_HW { ExternalAccessible := 'False'; ExternalVisible := 'False'} : Bool;   // Sturings hardware (PLC) in storing
         STS_KST_OPEN { ExternalAccessible := 'False'; ExternalVisible := 'False'} : Bool;   // TRUE = deur wegkantkast geopend
         STS_NEG { ExternalAccessible := 'False'; ExternalVisible := 'False'} : Bool;   // Spookrijder gedetecteerd
         STS_SOS { ExternalAccessible := 'False'; ExternalVisible := 'False'} : Bool;   // Snelheidsonderschrijding
         STS_STOP { ExternalAccessible := 'False'; ExternalVisible := 'False'} : Bool;   // Stilstand
      END_STRUCT;
   END_VAR
BEGIN

REGION Network 1: START
END_REGION

REGION Network 2: +++ Verkeersstatus +++
   // De door het detectiepunt geregistreerde verkeersstatus wordt doorgegeven aan 3B.
END_REGION

REGION Network 3: +++ Bewaking deur wegkantkast +++
   // De bewaking van de deur van de wegkantkast is enkel van toepassing voor detectiepunten die zich buiten de verkeerskoker bevinden en die aangesloten zijn via een wegkantkast behorende tot deelsysteem C403 (SOS).
END_REGION

REGION Network 4: +++ Storingen +++
   // Verzamelen storingsmeldingen.
END_REGION

REGION Network 5: Storing A001: Beveiliging aangesproken
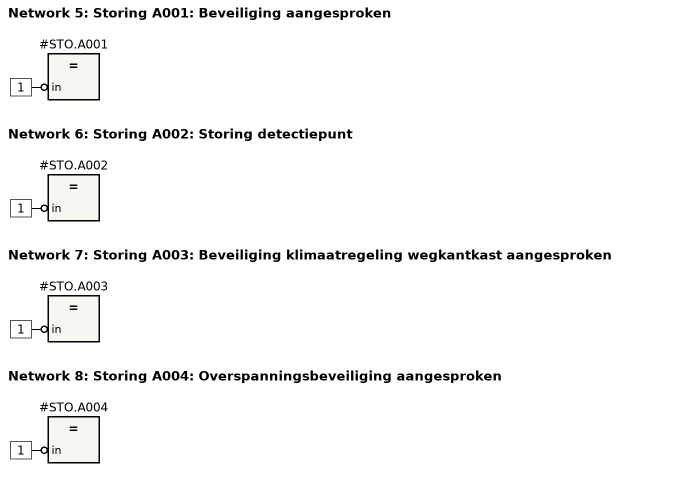
   #STO.A001 := NOT 1;
END_REGION

REGION Network 6: Storing A002: Storing detectiepunt
   #STO.A002 := NOT 1;
END_REGION

REGION Network 7: Storing A003: Beveiliging klimaatregeling wegkantkast aangesproken
   #STO.A003 := NOT 1;
END_REGION

REGION Network 8: Storing A004: Overspanningsbeveiliging aangesproken
   #STO.A004 := NOT 1;
END_REGION

REGION Network 9 (SCL): EINDE
   // Variabelen van intern scada rakvlak naar outputs copieren
   #VAR_IF_LVE.EXT_HW := #VAR.EXT_HW;
   #VAR_IF_LVE.STS_KST_OPEN := #VAR.STS_KST_OPEN;
   #VAR_IF_LVE.STS_NEG := #VAR.STS_NEG;
   #VAR_IF_LVE.STS_SOS := #VAR.STS_SOS;
   #VAR_IF_LVE.STS_STOP := #VAR.STS_STOP;
   #VAR_IF_LVE.STO := #STO;
END_REGION
END_FUNCTION_BLOCK

FUNCTION_BLOCK "TYPIC_C403_IF_SOS"   // FB118, FBD
TITLE = TYPIC_C403_IF_SOS: Snelheidsonderschrijding
{ S7_Optimized_Access := 'TRUE' }
AUTHOR : OCOTECH
FAMILY : Typical
NAME : C403.701
// Logisch Object Besturing: C403.701
// 
// Het doel van de IF SOS (SnelheidsOnderschrijdingsSysteem) is om de algemene gegevens te verwerken die ontvangen worden vanuit de interne sturing en via inputs.
// stored: MemoryReserve 10, SetENOAutomatically false
   VAR_INPUT
      EXT_HW { ExternalAccessible := 'False'; ExternalVisible := 'False'; ExternalWritable := 'False'} : Bool;   // Sturings hardware (PLC) bewaking (1 = OK)
      IN_AUT_C403 { ExternalAccessible := 'False'; ExternalVisible := 'False'; ExternalWritable := 'False'} : Bool;   // Beveiligingen: serie geschakelde terugmelding (1= OK)
      IN_STO { ExternalAccessible := 'False'; ExternalVisible := 'False'; ExternalWritable := 'False'} : Word;   // Algemene storingen
   END_VAR
   VAR_OUTPUT
      VAR_IF_SOS { ExternalAccessible := 'False'; ExternalVisible := 'False'; ExternalWritable := 'False'} : "C403_VAR_IF_SOS_TYPIC";   // Struct met alle variabelen naar de basisfunctie
   END_VAR
   VAR
      STO { ExternalWritable := 'False'} : Struct   // Storingen
         A001 : Bool;   // Beveiliging aangesproken
         A002 : Bool;   // SOS-detectie is over 60 m tot 150 m uitgevallen
         A003 : Bool;   // SOS-detectie is over meer dan 150 m uitgevallen
      END_STRUCT;
      VAR { ExternalWritable := 'False'} : Struct   // Variabelen
         EXT_HW { ExternalAccessible := 'False'; ExternalVisible := 'False'} : Bool;   // Sturings hardware (PLC) in storing
      END_STRUCT;
   END_VAR
BEGIN

REGION Network 1: START
END_REGION

REGION Network 2: +++ Storingen +++
   // Verzamelen storingsmeldingen.
END_REGION

REGION Network 3: Storing A001: Beveiliging aangesproken
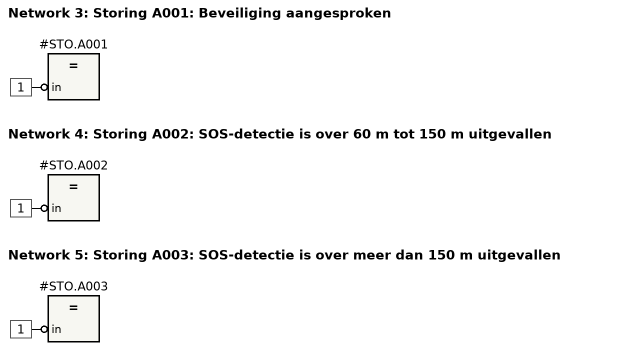
   #STO.A001 := NOT 1;
END_REGION

REGION Network 4: Storing A002: SOS-detectie is over 60 m tot 150 m uitgevallen
   #STO.A002 := NOT 1;
END_REGION

REGION Network 5: Storing A003: SOS-detectie is over meer dan 150 m uitgevallen
   #STO.A003 := NOT 1;
END_REGION

REGION Network 6 (SCL): EINDE
   // Variabelen van intern scada rakvlak naar outputs copieren
   #VAR_IF_SOS.EXT_HW := #VAR.EXT_HW;
   #VAR_IF_SOS.STO := #STO;
END_REGION
END_FUNCTION_BLOCK

FUNCTION_BLOCK "TYPIC_C403_SF_LVE"   // FB131, FBD
TITLE = TYPIC_C403_SF_LVE: Detectiepunt
{ S7_Optimized_Access := 'TRUE' }
AUTHOR : OCOTECH
FAMILY : Typical
NAME : C403.802
// Logisch Object Besturing: C403.802
// 
// De subfunctie detectiepunt verzorgt de bediening en sturing van een SOSodetectiepunt vanuit 3B en is tevens het raakvlak tussen 3B en de interne sturing van het detectiepunt.
// stored: MemoryReserve 10, SetENOAutomatically false
   VAR_INPUT
      CFG_STR { ExternalAccessible := 'False'; ExternalVisible := 'False'; ExternalWritable := 'False'} : USInt;   // Nummer van de rijstrook (1 = rechterrijstrook)
      CFG_NUM { ExternalAccessible := 'False'; ExternalVisible := 'False'; ExternalWritable := 'False'} : Int;   // Nummer van het detectiepunt op de rijstrook volgens rijrichting
      CFG_POS1 { ExternalAccessible := 'False'; ExternalVisible := 'False'; ExternalWritable := 'False'} : USInt;   // FO-naam van de verkeerskoker (of op- / afrit) waar het detectiepunt staat
      CFG_POS2 { ExternalAccessible := 'False'; ExternalVisible := 'False'; ExternalWritable := 'False'} : Real;   // Lengtepositie van het detectiepunt in de verkeerskoker
      CFG_LCK_AANT { ExternalAccessible := 'False'; ExternalVisible := 'False'; ExternalWritable := 'False'} : Int;   // Aantal stroomopwaartse detectiepunten waarin verkeerskundige meldingen onderdrukt worden
      STU_ALG_LCK_SIG { ExternalAccessible := 'False'; ExternalVisible := 'False'; ExternalWritable := 'False'} : USInt;   // Onderdruk alarmen
   END_VAR
   VAR_OUTPUT
      VAR_LVE { ExternalAccessible := 'False'; ExternalVisible := 'False'; ExternalWritable := 'False'} : "C403_VAR_LVE_TYPIC";   // Struct met alle variabelen van de SOS-sectie
   END_VAR
   VAR_IN_OUT
      STU_LVE : "C403_STU_LVE_TYPIC";   // Sturing Detectiepunten
      VAR_IF_LVE : "C403_VAR_IF_LVE_TYPIC";   // Struct met alle variabelen ontvangen van de functie (IF) in de interne sturing van het afsluitsysteem
   END_VAR
   VAR
      BED : Struct   // Bedieningen
         OBS : Struct   // SOS-sectie aan- of uitschakelen
            X : "UDT_BED_ALG";
            KNOP { S7_SetPoint := 'True'} : Array[0..1] of "UDT_BED_KNOP";
         END_STRUCT;
         VGV_SIG : Struct   // Signalering verkeerskundige alarmen vrijgeven of onderdrukken
            X : "UDT_BED_ALG";
            KNOP { S7_SetPoint := 'True'} : Array[0..1] of "UDT_BED_KNOP";
         END_STRUCT;
      END_STRUCT;
      BED_OBS { ExternalWritable := 'False'} : "TYPIC_HF_BED_ALG_KNOP";   // SOS-sectie aan- of uitschakelen
      BED_VGV_SIG { ExternalWritable := 'False'} : "TYPIC_HF_BED_ALG_KNOP";   // Signalering verkeerskundige alarmen vrijgeven of onderdrukken
      SIG { ExternalWritable := 'False'} : Struct   // Signaleringen
         AA01 : Bool;   // Detectiepunt niet observeerbaar
         AA02 : Bool;   // Storing algemeen
         AA03 : Bool;   // Deur wegkantkast geopend
         AV01 : Bool;   // Stilstand gedetecteerd
         AV02 : Bool;   // Snelheidsonderschrijding gedetecteerd
         AV03 : Bool;   // Spookrijder gedetecteerd
         A001 : Bool;   // Beveiliging aangesproken
         A002 : Bool;   // Storing detectiepunt
         A003 : Bool;   // Beveiliging klimaatregeling wegkantkast aangesproken
         A004 : Bool;   // Overspanningsbeveiliging aangesproken
      END_STRUCT;
      VAR { ExternalWritable := 'False'} : Struct   // Variabelen
         STS_STOP : USInt;   // Stilstand gedetecteerd
         STS_SOS : USInt;   // Snelheidsonderschrijding gedetecteerd
         RNO : USInt;   // Reden niet bestuurbaar
         VGV_SIG_VOP : Bool;   // TRUE = Signaleringen vrijgegeven voor verkeersoperator FALSE = Onderdrukt
         MEM_STS_STOP { ExternalAccessible := 'False'; ExternalVisible := 'False'} : Bool;   // TRUE = Stilstand gedetecteerd
         MEM_STS_SOS { ExternalAccessible := 'False'; ExternalVisible := 'False'} : Bool;   // TRUE = Snelheidsonderschrijding gedetecteerd
         STS_STOP_NEW { ExternalAccessible := 'False'; ExternalVisible := 'False'} : Bool;   // TRUE = Nieuwe detectie Stilstand
         STS_SOS_NEW { ExternalAccessible := 'False'; ExternalVisible := 'False'} : Bool;   // TRUE = Nieuwe detectie snelheidsonderschrijding
         LCK_STOP { ExternalAccessible := 'False'; ExternalVisible := 'False'} : Bool;   // TRUE = Onderdrukken signalering stilstand
         LCK_SOS { ExternalAccessible := 'False'; ExternalVisible := 'False'} : Bool;   // TRUE = Onderdrukken signalering SOS
         BSC : USInt;   // Beschikbaarheid
         STS_NEG : USInt;   // Spookrijder gedetecteerd
         OBS { ExternalAccessible := 'False'; ExternalVisible := 'False'} : USInt;   // Observeerbaarheid
         SIG_AV01 { ExternalAccessible := 'False'; ExternalVisible := 'False'} : USInt;   // Signalering Stilstand gedetecteerd actief
         SIG_AV02 { ExternalAccessible := 'False'; ExternalVisible := 'False'} : USInt;   // Signalering Snelheidsonderschrijding actief
         POS { ExternalAccessible := 'False'; ExternalVisible := 'False'} : Bool;   // Positie van het detectiepunt
      END_STRUCT;
      HF_BST_OBS { ExternalAccessible := 'False'; ExternalVisible := 'False'; ExternalWritable := 'False'} : "TYPIC_HF_BST_OBS";   // Hulp functie besturing
   END_VAR
   // // BED.OBS.KNOP[0] : InDienst
   // // BED.OBS.KNOP[1] : UitDienst
   // // BED.VGV_SIG.KNOP[0] : Ja
   // // BED.VGV_SIG.KNOP[1] : Onderdrukt
BEGIN

REGION Network 1: START
END_REGION

REGION Network 2: +++ Bedieningen +++
   // Vrijgave en verwerking van de bedieningen (centrale en lokale bediening). De bedienwaardes worden daarna in de verdere deelfunctionaliteiten gebruikt.
END_REGION

REGION Network 3: Knoppen BED_OBS(SOS-sectie aan- of uitschakelen)
   // Waardes en vrijge van de knoppen BED_OBS
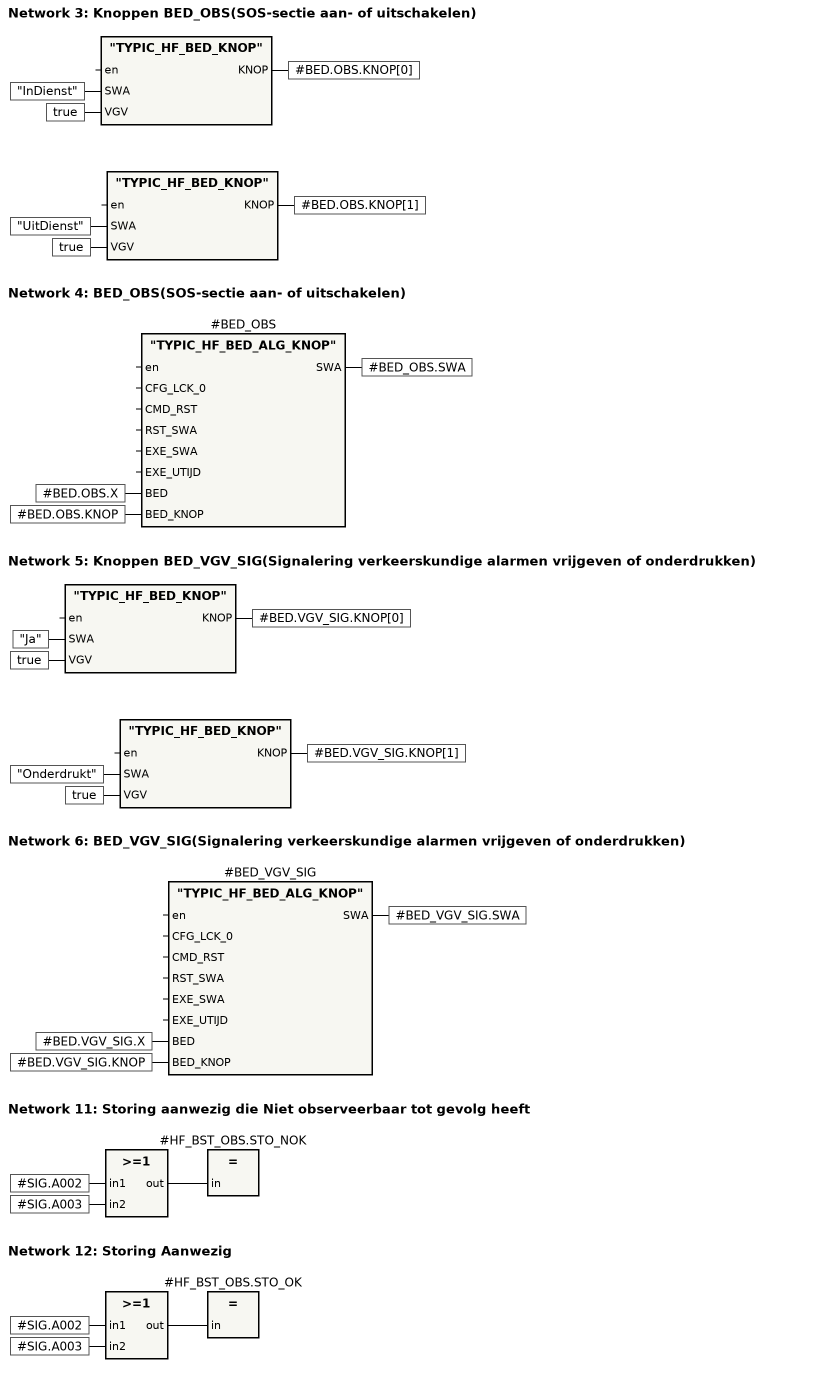
   "TYPIC_HF_BED_KNOP"(SWA := "InDienst", VGV := true, KNOP => #BED.OBS.KNOP[0]);
   "TYPIC_HF_BED_KNOP"(SWA := "UitDienst", VGV := true, KNOP => #BED.OBS.KNOP[1]);
END_REGION

REGION Network 4: BED_OBS(SOS-sectie aan- of uitschakelen)
   // Verwerking BED_OBS
   #BED_OBS(BED := #BED.OBS.X, BED_KNOP := #BED.OBS.KNOP, SWA => #BED_OBS.SWA);   // "TYPIC_HF_BED_ALG_KNOP"
END_REGION

REGION Network 5: Knoppen BED_VGV_SIG(Signalering verkeerskundige alarmen vrijgeven of onderdrukken)
   // Waardes en vrijge van de knoppen BED_VGV_SIG
   "TYPIC_HF_BED_KNOP"(SWA := "Ja", VGV := true, KNOP => #BED.VGV_SIG.KNOP[0]);
   "TYPIC_HF_BED_KNOP"(SWA := "Onderdrukt", VGV := true, KNOP => #BED.VGV_SIG.KNOP[1]);
END_REGION

REGION Network 6: BED_VGV_SIG(Signalering verkeerskundige alarmen vrijgeven of onderdrukken)
   // Verwerking BED_VGV_SIG
   #BED_VGV_SIG(BED := #BED.VGV_SIG.X, BED_KNOP := #BED.VGV_SIG.KNOP, SWA => #BED_VGV_SIG.SWA);   // "TYPIC_HF_BED_ALG_KNOP"
END_REGION

REGION Network 7: +++ Verwerken verkeersstatus +++
   // De ontvangen verkeersstatus vanuit de interne sturing omzetten naar variabelen
END_REGION

REGION Network 8: +++ Voorwaarden signalering stilstand +++
   // Een stilstand wordt gesignaleerd als bij opkomen van de detectie stilstand er geen onderdrukking is. Signaleringen kunnen onderdrukt worden als er detectiepunten stroomafwaarts reeds een stilstand signaleren.
END_REGION

REGION Network 9: +++ Voorwaarden signalering snelheidsonderschrijding +++
   // Een snelheidsonderschrijding wordt gesignaleerd als bij opkomen van de detectie snelheidsonderschrijding er geen onderdrukking is. Signaleringen kunnen onderdrukt worden als er detectiepunten stroomafwaarts reeds een snelheidsonderschrijding signaleren.
END_REGION

REGION Network 10: +++ Signaleringen en observeerbaarheid +++
   // Aanmaken signaleringen, bepalen observeerbaarheid (observeerbaar / niet observeerbaar) en bepalen reden niet observeerbaar.
END_REGION

REGION Network 11: Storing aanwezig die Niet observeerbaar tot gevolg heeft
   // OR-verknoping van alle storingen om input STO_BST_NOK van de hulpfunctie "Observeerbaarheid en algemene signlaring"
   #HF_BST_OBS.STO_NOK := #SIG.A002 OR #SIG.A003;
END_REGION

REGION Network 12: Storing Aanwezig
   // OR-verknoping van alle storingen om input STO_BST_OK van de hulpfunctie "Observeerbaarheid en algemene signlaring"
   #HF_BST_OBS.STO_OK := #SIG.A002 OR #SIG.A003;
END_REGION

REGION Network 13: Hulpfunctie "Observeerbaarheid en algemene signalering "
   // Bepalen variabele "Observeerbaarheid" en "reden niet Observeerbaarheid", Signaleringen "Observeerbaarheid" en "algmene storing".
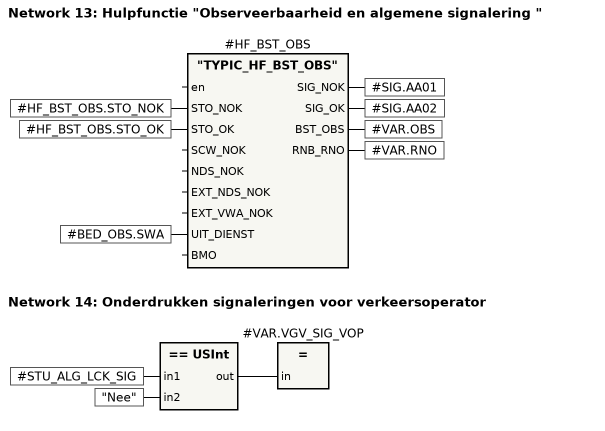
   #HF_BST_OBS(STO_NOK := #HF_BST_OBS.STO_NOK,   // "TYPIC_HF_BST_OBS"
               STO_OK := #HF_BST_OBS.STO_OK,
               UIT_DIENST := #BED_OBS.SWA,
               SIG_NOK => #SIG.AA01,
               SIG_OK => #SIG.AA02,
               BST_OBS => #VAR.OBS,
               RNB_RNO => #VAR.RNO);
END_REGION

REGION Network 14: Onderdrukken signaleringen voor verkeersoperator
   // Via de variabele VGV_SIG_VOP wordt aan IRIS SCADA doorgegeven of signaleringen (bestemd voor de verkeersoperator) van de deze functie zichtbaar (of onderdrukt) moeten zijn.
   #VAR.VGV_SIG_VOP := #STU_ALG_LCK_SIG = "Nee";
END_REGION

REGION Network 15: +++ Bepalen beschikbaarheidsstatus +++
   // Beschikbaarheidsstatus (Uit Dienst / beschikbaar / beperkt beschikbaar / niet beschikbaar) bepalen.
END_REGION

REGION Network 16 (SCL): Beschikbaarheidsstatus bepalen
   IF 
       //voorwaarden "Niet beschikbaar"
       TRUE
   THEN
       //Beschikbaarheidsstatus = Niet Beschikbaar
       #VAR.BSC:= "NietBeschikbaar";
   ELSIF
       //voorwaarden "Beperkt beschikbaar"
       TRUE
   THEN
       //Beschikbaarheidsstatus = Beperkt Beschikbaar
       #VAR.BSC:= "Beperkt";
   ELSE
       //Beschikbaarheidsstatus = Beschikbaar
       #VAR.BSC:= "Beschikbaar";
   END_IF;
END_REGION

REGION Network 17: +++ Verwerken configuraties +++
   // De configuraties verwerken naar variabelen.
END_REGION

REGION Network 18 (SCL): EINDE
   // Variabelen van intern scada rakvlak naar outputs copieren
   #VAR_LVE.BSC := #VAR.BSC;
   #VAR_LVE.STS_NEG := #VAR.STS_NEG;
   #VAR_LVE.OBS := #VAR.OBS;
   #VAR_LVE.SIG_AV01 := #VAR.SIG_AV01;
   #VAR_LVE.SIG_AV02 := #VAR.SIG_AV02;
   #VAR_LVE.POS := #VAR.POS;
END_REGION
END_FUNCTION_BLOCK

FUNCTION_BLOCK "TYPIC_C406_BF_CAD"   // FB10, FBD
TITLE = TYPIC_C406_BF_CAD: CaDo Tunnel
{ S7_Optimized_Access := 'TRUE' }
AUTHOR : OCOTECH
FAMILY : Typical
NAME : C406.801
// Logisch Object Besturing: C406.801
// 
// Het doel van de BF CAD (CaDo Tunnel) is om de algemene sturing te voorzien van de calamiteiten doorsteek.
// 
// De algemene sturing omvat het weergeven van de algemene toestand en het openen en sluiten van calamiteiten doorsteek ten behoeve van de hulpdiensten en werkverkeer.
// stored: MemoryReserve 10, SetENOAutomatically false
   VAR_INPUT
      STU_AUT_CMD { ExternalAccessible := 'False'; ExternalVisible := 'False'; ExternalWritable := 'False'} : USInt;   // Sturing calamiteitendoorsteek algemeen
      STU_ALG_LCK_SIG { ExternalAccessible := 'False'; ExternalVisible := 'False'; ExternalWritable := 'False'} : USInt;   // Onderdruk alarmen
      STU_CAD_LCK_SIG { ExternalAccessible := 'False'; ExternalVisible := 'False'; ExternalWritable := 'False'} : USInt;   // Onderdruk alarm Cado niet dicht
      CFG_TST_UTYD { ExternalAccessible := 'False'; ExternalVisible := 'False'; ExternalWritable := 'False'} : Time;   // Maximale transitietijd stand verandering calamiteitendoorsteek (transitiestatus niet bereikt)
      CFG_TST_OK_TYD { ExternalAccessible := 'False'; ExternalVisible := 'False'; ExternalWritable := 'False'} : Time;   // Stabilisatietijd voor de toestand OK (bereikt)
   END_VAR
   VAR_OUTPUT
      STU_CAD_CMD { ExternalAccessible := 'False'; ExternalVisible := 'False'; ExternalWritable := 'False'} : USInt;   // Sturing CaDo algemeen
   END_VAR
   VAR_IN_OUT
      VAR_CAD : Array[0..1] of Bool;   // Array met alle calamiteitendoorsteken, met alle variabelen van de calamiteitendoorsteek
   END_VAR
   VAR
      BED : Struct   // Bedieningen
         ALG : Struct   // Gewenste stand
            X : "UDT_BED_ALG";
            KNOP { S7_SetPoint := 'True'} : Array[0..3] of "UDT_BED_KNOP";
         END_STRUCT;
      END_STRUCT;
      BED_ALG { ExternalWritable := 'False'} : "TYPIC_HF_BED_ALG_KNOP";   // Gewenste stand
      SIG { ExternalWritable := 'False'} : Struct   // Signaleringen
         AA01 : Bool;   // Gewenste stand niet bereikt
         AB01 : Bool;   // CaDo niet beschikbaar
         AB02 : Bool;   // CaDo beperkt beschikbaar
         AV01 : Bool;   // CaDo niet dicht
      END_STRUCT;
      VAR { ExternalWritable := 'False'} : Struct   // Variabelen
         BMO : USInt;   // Bedieningsmode
         TST_BWA : USInt;   // De status van de transitie van de CaDo
         BSC : USInt;   // Geeft de beschikbaarheidsstatus van de CaDo aan
         CAD_SWA : USInt;   // Doelstand CaDo
         CAD_BWA : USInt;   // Werkelijke stand CaDo
         VGV_SIG_VOP : Bool;   // TRUE = Signaleringen vrijgegeven voor verkeersoperator FALSE = Onderdrukt
      END_STRUCT;
      HF_TST { ExternalAccessible := 'False'; ExternalVisible := 'False'; ExternalWritable := 'False'} : "TYPIC_HF_TST";   // Hulpfunctie transitiestatus
   END_VAR
   // // BED.ALG.KNOP[0] : Auto
   // // BED.ALG.KNOP[1] : Open
   // // BED.ALG.KNOP[2] : Dicht
   // // BED.ALG.KNOP[3] : Stop
BEGIN

REGION Network 1: START
END_REGION

REGION Network 2: +++ Bedieningen +++
   // Vrijgave en verwerking van de bedieningen (centrale en lokale bediening). De bedienwaardes worden daarna in de verdere deelfunctionaliteiten gebruikt.
END_REGION

REGION Network 3: Knoppen BED_ALG(Gewenste stand)
   // Waardes en vrijge van de knoppen BED_ALG
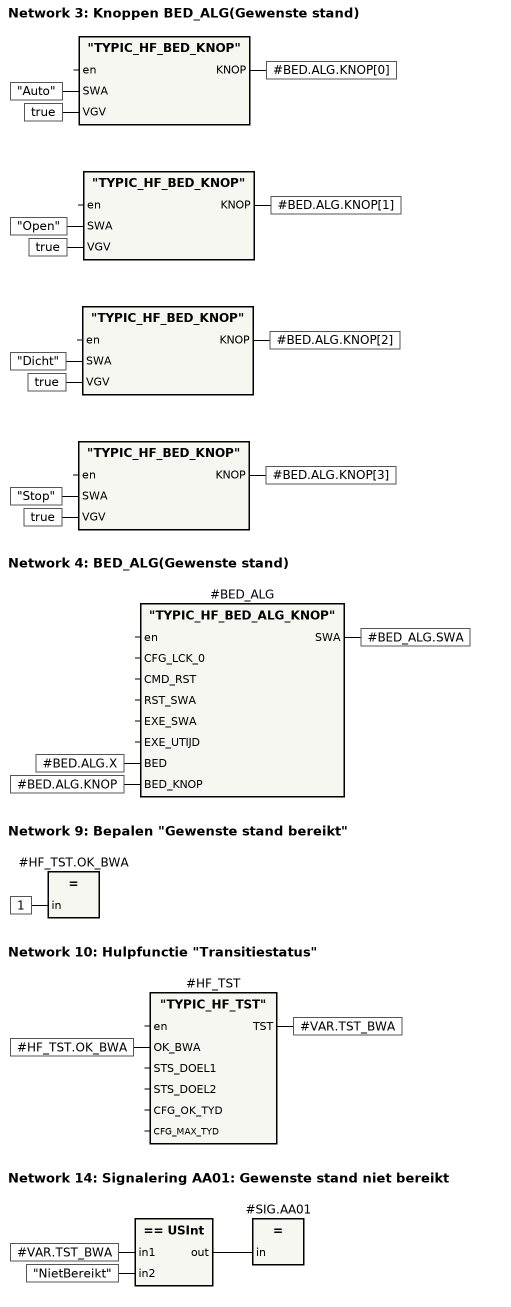
   "TYPIC_HF_BED_KNOP"(SWA := "Auto", VGV := true, KNOP => #BED.ALG.KNOP[0]);
   "TYPIC_HF_BED_KNOP"(SWA := "Open", VGV := true, KNOP => #BED.ALG.KNOP[1]);
   "TYPIC_HF_BED_KNOP"(SWA := "Dicht", VGV := true, KNOP => #BED.ALG.KNOP[2]);
   "TYPIC_HF_BED_KNOP"(SWA := "Stop", VGV := true, KNOP => #BED.ALG.KNOP[3]);
END_REGION

REGION Network 4: BED_ALG(Gewenste stand)
   // Verwerking BED_ALG
   #BED_ALG(BED := #BED.ALG.X, BED_KNOP := #BED.ALG.KNOP, SWA => #BED_ALG.SWA);   // "TYPIC_HF_BED_ALG_KNOP"
END_REGION

REGION Network 5: +++ Bedieningsmode +++
   // Bedieningsmode (Auto / Manueel ) bepalen.
END_REGION

REGION Network 6: +++ Bepalen gewenst stand +++
   // Bepalen van de gewenste stand (Open / Dicht / Stop)
END_REGION

REGION Network 7: +++ Bepalen werkelijke stand +++
   // Bepalen van de werkelijke stand (Open / Dicht / DichtVerlaten / Onbepaald) aan de hand van positiestatus van de calamiteitendoorsteken.
END_REGION

REGION Network 8: +++ Bepalen transitiestatus +++
   // Transitiestatus (bereikt / niet bereikt / in transitie) bepalen.
END_REGION

REGION Network 9: Bepalen "Gewenste stand bereikt"
   // Bepalen of de actuele stand in overeenstemming is met de gewenste stand
   #HF_TST.OK_BWA := 1;
END_REGION

REGION Network 10: Hulpfunctie "Transitiestatus"
   // De transitiestatus geeft de relatie tussen een gewenste stand (van een functionaliteit) en de actuele stand aan.
   #HF_TST(OK_BWA := #HF_TST.OK_BWA, TST => #VAR.TST_BWA);   // "TYPIC_HF_TST"
END_REGION

REGION Network 11: +++ Bepalen beschikbaarheidsstatus +++
   // Beschikbaarheidsstatus (beschikbaar / beperkt beschikbaar / niet beschikbaar) bepalen.
END_REGION

REGION Network 12 (SCL): Beschikbaarheidsstatus bepalen
   IF 
       //voorwaarden "Niet beschikbaar"
       TRUE
   THEN
       //Beschikbaarheidsstatus = Niet Beschikbaar
       #VAR.BSC:= "NietBeschikbaar";
   ELSIF
       //voorwaarden "Beperkt beschikbaar"
       TRUE
   THEN
       //Beschikbaarheidsstatus = Beperkt Beschikbaar
       #VAR.BSC:= "Beperkt";
   ELSE
       //Beschikbaarheidsstatus = Beschikbaar
       #VAR.BSC:= "Beschikbaar";
   END_IF;
END_REGION

REGION Network 13: +++ Signaleringen +++
   // Aanmaken signaleringen.
END_REGION

REGION Network 14: Signalering AA01: Gewenste stand niet bereikt
   #SIG.AA01 := #VAR.TST_BWA = "NietBereikt";
END_REGION

REGION Network 15: Signalering AB01 : Niet Beschikbaar
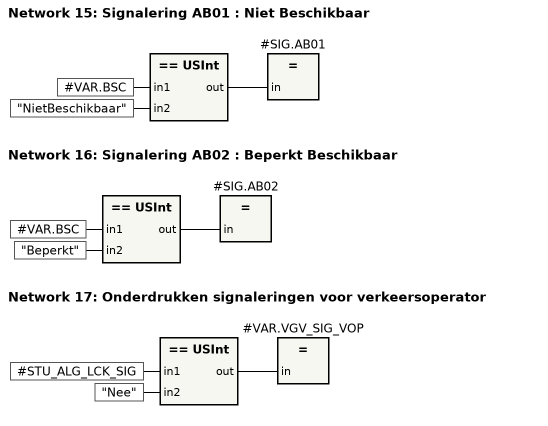
   #SIG.AB01 := #VAR.BSC = "NietBeschikbaar";
END_REGION

REGION Network 16: Signalering AB02 : Beperkt Beschikbaar
   #SIG.AB02 := #VAR.BSC = "Beperkt";
END_REGION

REGION Network 17: Onderdrukken signaleringen voor verkeersoperator
   // Via de variabele VGV_SIG_VOP wordt aan IRIS SCADA doorgegeven of signaleringen (bestemd voor de verkeersoperator) van de deze functie zichtbaar (of onderdrukt) moeten zijn.
   #VAR.VGV_SIG_VOP := #STU_ALG_LCK_SIG = "Nee";
END_REGION

REGION Network 18: +++ Sturingen +++
   // Individuele commandos uitsturen naar iedere calamiteiten doorsteek om te openen en te sluiten.
END_REGION

REGION Network 19: EINDE
   // Variabelen van intern scada rakvlak naar outputs copieren
END_REGION
END_FUNCTION_BLOCK

FUNCTION_BLOCK "TYPIC_C501_IF_ABP"   // FB6, FBD
TITLE = TYPIC_C501_IF_ABP: Automatische Brandbluspomp
{ S7_Optimized_Access := 'TRUE' }
AUTHOR : OCOTECH
FAMILY : Typical
NAME : C501.708
// Logisch Object Besturing: C501.708
// 
// De interne functie brandbluspomp verzorgt de interne besturing, bewaking en fysieke aansturing van een automatische brandbluspomp behorend tot de brandblusinstallatie.
// stored: MemoryReserve 10, SetENOAutomatically false
   VAR_INPUT
      PULS_100ms { ExternalAccessible := 'False'; ExternalVisible := 'False'; ExternalWritable := 'False'} : Bool;   // Puls, 1 PLC-cyclus hoog, 1 keer per 100 ms
      PULS_1s { ExternalAccessible := 'False'; ExternalVisible := 'False'; ExternalWritable := 'False'} : Bool;   // Puls, 1 PLC-cyclus hoog, 1 keer per seconde
      EXT_HW { ExternalAccessible := 'False'; ExternalVisible := 'False'; ExternalWritable := 'False'} : Bool;   // Sturings hardware (PLC) bewaking (1 = OK)
      IN_HND { ExternalAccessible := 'False'; ExternalVisible := 'False'; ExternalWritable := 'False'} : Bool;   // Terugmelding aansturing via hand (hardware)
      IN_AAN { ExternalAccessible := 'False'; ExternalVisible := 'False'; ExternalWritable := 'False'} : Bool;   // Terugmelding aansturing
      IN_SNE { ExternalAccessible := 'False'; ExternalVisible := 'False'; ExternalWritable := 'False'} : Bool;   // Actuele snelheid pomp
      IN_AUT_C501 { ExternalAccessible := 'False'; ExternalVisible := 'False'; ExternalWritable := 'False'} : Bool;   // Beveiligingen: serie geschakelde terugmelding (1= OK)
      IN_AUT { ExternalAccessible := 'False'; ExternalVisible := 'False'; ExternalWritable := 'False'} : Bool;   // Status thermische beveiliging (1 = OK)
      IN_PTC { ExternalAccessible := 'False'; ExternalVisible := 'False'; ExternalWritable := 'False'} : Bool;   // Detectie hoge temperatuur in de wikkelingen van de motor (1 = OK)
      IN_SCW { ExternalAccessible := 'False'; ExternalVisible := 'False'; ExternalWritable := 'False'} : Bool;   // Werkschakelaar (1 = Aan)
      IN_STO { ExternalAccessible := 'False'; ExternalVisible := 'False'; ExternalWritable := 'False'} : Bool;   // Status Frequentieomvormer (1 = OK)
      IN_DME_STO { ExternalAccessible := 'False'; ExternalVisible := 'False'; ExternalWritable := 'False'} : Bool;   // Filterbewaking (1= OK / 0 = Vervuild)
      IN_STS1 { ExternalAccessible := 'False'; ExternalVisible := 'False'; ExternalWritable := 'False'} : Bool;   // Status motorlade ingeschakeld
      IN_STS2 { ExternalAccessible := 'False'; ExternalVisible := 'False'; ExternalWritable := 'False'} : Bool;   // Status motorlade in test
      IN_STS3 { ExternalAccessible := 'False'; ExternalVisible := 'False'; ExternalWritable := 'False'} : Bool;   // Status motorlade uitgereden
      IN_STR1 { ExternalAccessible := 'False'; ExternalVisible := 'False'; ExternalWritable := 'False'} : Int;   // Analoge meting ventilator fasestroom 1
      IN_STR2 { ExternalAccessible := 'False'; ExternalVisible := 'False'; ExternalWritable := 'False'} : Int;   // Analoge meting ventilator fasestroom 2
      IN_STR3 { ExternalAccessible := 'False'; ExternalVisible := 'False'; ExternalWritable := 'False'} : Int;   // Analoge meting ventilator fasestroom 3
      IN_TRL { ExternalAccessible := 'False'; ExternalVisible := 'False'; ExternalWritable := 'False'} : Bool;   // Trillingsdetectie (1 = Geen trillingen)
      CFG_MIN_SNE { ExternalAccessible := 'False'; ExternalVisible := 'False'; ExternalWritable := 'False'} : Real;   // Minimale stuursnelheid automatische brandbluspompen
      CFG_TYD_FB { ExternalAccessible := 'False'; ExternalVisible := 'False'; ExternalWritable := 'False'} : Time;   // Vertragingstijd storing foute terugmelding
      CFG_TYD_TRL { ExternalAccessible := 'False'; ExternalVisible := 'False'; ExternalWritable := 'False'} : Time;   // Vertragingstijd storing onbalans
      CFG_TRL_MAX { ExternalAccessible := 'False'; ExternalVisible := 'False'; ExternalWritable := 'False'} : Real;   // Hoogste waarde scalering trillingsmeting
      CFG_TRL_MIN { ExternalAccessible := 'False'; ExternalVisible := 'False'; ExternalWritable := 'False'} : Real;   // Laagste waarde scalering trillingsmeting
      CFG_TRL_HOOG { ExternalAccessible := 'False'; ExternalVisible := 'False'; ExternalWritable := 'False'} : Real;   // Schakeldrempel hoog trillingsmeting (onbalans)
      CFG_TYD_RUN { ExternalAccessible := 'False'; ExternalVisible := 'False'; ExternalWritable := 'False'} : LInt;   // Minimale draaitijd om melding onderhoud nodig te resetten
      CFG_TYD_STOP { ExternalAccessible := 'False'; ExternalVisible := 'False'; ExternalWritable := 'False'} : LInt;   // Stilstandstijd die melding onderhoud nodig activeert
      CFG_TYD_MAX { ExternalAccessible := 'False'; ExternalVisible := 'False'; ExternalWritable := 'False'} : Int;   // Tijdsduur draaitijd overschrijding pomp
   END_VAR
   VAR_OUTPUT
      VAR_IF_ABP { ExternalAccessible := 'False'; ExternalVisible := 'False'; ExternalWritable := 'False'} : "C501_VAR_IF_ABP_TYPIC";   // Struct met alle variabelen naar bovenliggende functies
      OUT_AAN { ExternalAccessible := 'False'; ExternalVisible := 'False'; ExternalWritable := 'False'} : Bool;   // Aansturen pomp
      OUT_RES { ExternalAccessible := 'False'; ExternalVisible := 'False'; ExternalWritable := 'False'} : Bool;   // Reset Frequentieomvormer
      OUT_SNE { ExternalAccessible := 'False'; ExternalVisible := 'False'; ExternalWritable := 'False'} : Int;   // Sturing snelheid pomp
   END_VAR
   VAR_IN_OUT
      STU_IF_ABP : "C501_STU_IF_ABP_TYPIC";   // Struct met alle sturingen van de subfunctie (SF) pomp van 3B
   END_VAR
   VAR
      BED : Struct   // Bedieningen
         REM : Bool;   // Bediening om pomp in Remote te schakelen (indien IN_HND = 0)
         FWD : Bool;   // Bediening om pomp in hand te schakelen en te starten
         STOP : Bool;   // Bediening om pomp in hand te schakelen en te stoppen
         RES : Bool;   // Reset storingen
         SNE : Real;   // Bediening snelheid pomp
      END_STRUCT;
      STO { ExternalWritable := 'False'} : Struct   // Storingen
         A001 : Bool;   // Beveiliging aangesproken
         A002 : Bool;   // Storing van de motorbeveiliging van de pomp
         A003 : Bool;   // Storing Frequentieomvormer
         A004 : Bool;   // Te hoge temperatuur in de motorwikkelingen
         A005 : Bool;   // De pomp is in onbalans
         A006 : Bool;   // Motorlade uitgeschakeld
         A007 : Bool;   // Motorlade in test
         A008 : Bool;   // Motorlade uitgereden
         A009 : Bool;   // Fout stroommeting fase 1
         A010 : Bool;   // Fout stroommeting fase 2
         A011 : Bool;   // Fout stroommeting fase 3
         A012 : Bool;   // Filter vervuild
         AT01 : Bool;   // Discordantie motor: terugmelding niet ontvangen
         AT02 : Bool;   // Discordantie motor: terugmelding blijft aanwezig
         M001 : Bool;   // Werkschakelaar uitgeschakeld
         M002 : Bool;   // Melding: Pomp heeft te lang niet gedraaid. Periodiek onderhoud nodig
         M003 : Bool;   // Melding: Draaitijd overschrijding
      END_STRUCT;
      VAR { ExternalWritable := 'False'} : Struct   // Variabelen
         STS_AAN : Bool;   // Pomp draait
         STS_SNE : Real;   // Actuele snelheid pomp
         BMO_HAND : Bool;   // Pomp in hand geschakeld
         TYD_TOT_AAN { ExternalAccessible := 'False'; ExternalVisible := 'False'} : LInt;   // Totaal aantal draaiuren (in seconden)
         TYD_TOT_AAN_UUR { ExternalAccessible := 'False'; ExternalVisible := 'False'} : LInt;   // Totaal aantal draaiuren (in uren)
         TYD_AAN { ExternalAccessible := 'False'; ExternalVisible := 'False'} : Int;   // Aantal seconden dat pomp aangeschakeld is
         TYD_UIT { ExternalAccessible := 'False'; ExternalVisible := 'False'} : Int;   // Aantal seconden dat pomp uitgeschakeld is
         ENE_MWA1 { ExternalAccessible := 'False'; ExternalVisible := 'False'} : Real;   // Stroommeting fase 1
         ENE_MWA2 { ExternalAccessible := 'False'; ExternalVisible := 'False'} : Real;   // Stroommeting fase 2
         ENE_MWA3 { ExternalAccessible := 'False'; ExternalVisible := 'False'} : Real;   // Stroommeting fase 3
         EXT_HW { ExternalAccessible := 'False'; ExternalVisible := 'False'} : Bool;   // Sturings hardware (PLC) in storing
      END_STRUCT;
   END_VAR
BEGIN

REGION Network 1: START
END_REGION

REGION Network 2: +++ Metingen +++
   // Inlezen van de 3 stroommetingen van iedere fase van de motor.
END_REGION

REGION Network 3: +++ Storingen +++
   // Verwerken van de storingsmeldingen (inputs).
END_REGION

REGION Network 4: Storing A001: Beveiliging aangesproken
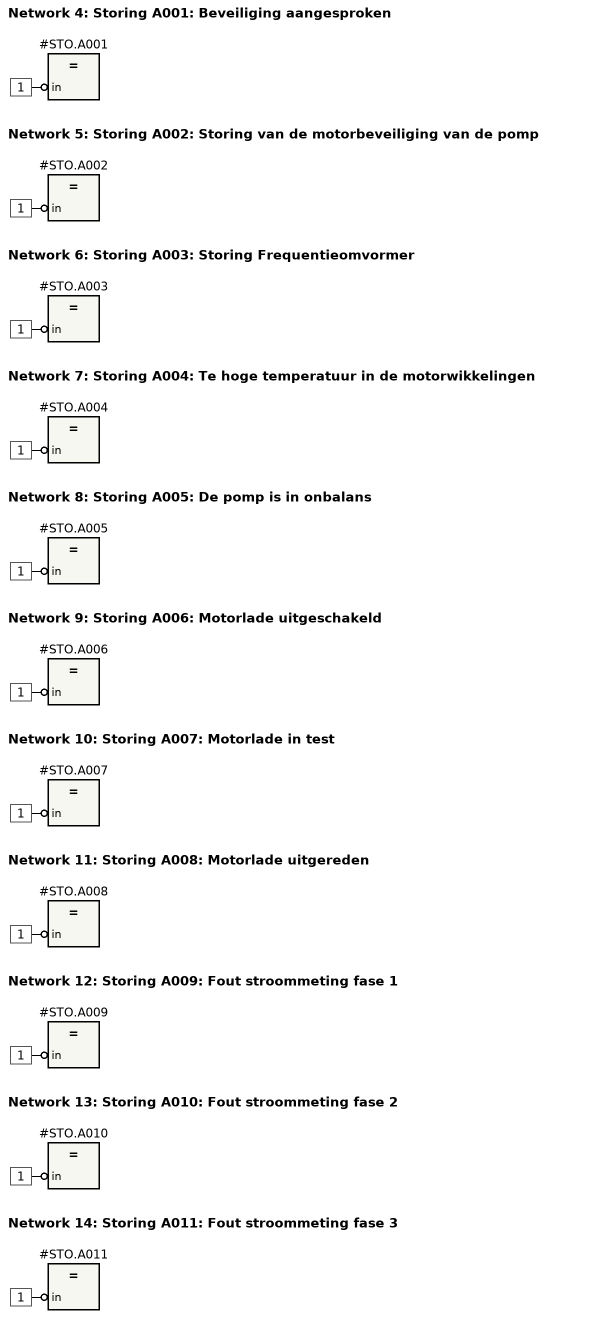
   #STO.A001 := NOT 1;
END_REGION

REGION Network 5: Storing A002: Storing van de motorbeveiliging van de pomp
   #STO.A002 := NOT 1;
END_REGION

REGION Network 6: Storing A003: Storing Frequentieomvormer
   #STO.A003 := NOT 1;
END_REGION

REGION Network 7: Storing A004: Te hoge temperatuur in de motorwikkelingen
   #STO.A004 := NOT 1;
END_REGION

REGION Network 8: Storing A005: De pomp is in onbalans
   #STO.A005 := NOT 1;
END_REGION

REGION Network 9: Storing A006: Motorlade uitgeschakeld
   #STO.A006 := NOT 1;
END_REGION

REGION Network 10: Storing A007: Motorlade in test
   #STO.A007 := NOT 1;
END_REGION

REGION Network 11: Storing A008: Motorlade uitgereden
   #STO.A008 := NOT 1;
END_REGION

REGION Network 12: Storing A009: Fout stroommeting fase 1
   #STO.A009 := NOT 1;
END_REGION

REGION Network 13: Storing A010: Fout stroommeting fase 2
   #STO.A010 := NOT 1;
END_REGION

REGION Network 14: Storing A011: Fout stroommeting fase 3
   #STO.A011 := NOT 1;
END_REGION

REGION Network 15: Storing A012: Filter vervuild
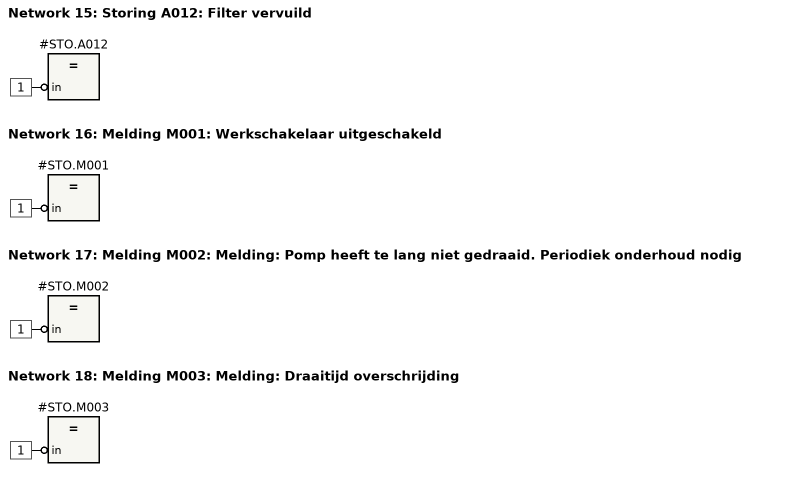
   #STO.A012 := NOT 1;
END_REGION

REGION Network 16: Melding M001: Werkschakelaar uitgeschakeld
   #STO.M001 := NOT 1;
END_REGION

REGION Network 17: Melding M002: Melding: Pomp heeft te lang niet gedraaid. Periodiek onderhoud nodig
   #STO.M002 := NOT 1;
END_REGION

REGION Network 18: Melding M003: Melding: Draaitijd overschrijding
   #STO.M003 := NOT 1;
END_REGION

REGION Network 19: +++ Motorsturing +++
   // Aansturen en bewaking van de motor.
END_REGION

REGION Network 20: +++ Urentellers +++
   // Tellen van de tijdsduur dat motor draait of stilstaat.
END_REGION

REGION Network 21 (SCL): EINDE
   // Variabelen van intern scada rakvlak naar outputs copieren
   #VAR_IF_ABP.STS_AAN := #VAR.STS_AAN;
   #VAR_IF_ABP.STS_SNE := #VAR.STS_SNE;
   #VAR_IF_ABP.BMO_HAND := #VAR.BMO_HAND;
   #VAR_IF_ABP.TYD_TOT_AAN := #VAR.TYD_TOT_AAN;
   #VAR_IF_ABP.TYD_TOT_AAN_UUR := #VAR.TYD_TOT_AAN_UUR;
   #VAR_IF_ABP.TYD_AAN := #VAR.TYD_AAN;
   #VAR_IF_ABP.TYD_UIT := #VAR.TYD_UIT;
   #VAR_IF_ABP.ENE_MWA1 := #VAR.ENE_MWA1;
   #VAR_IF_ABP.ENE_MWA2 := #VAR.ENE_MWA2;
   #VAR_IF_ABP.ENE_MWA3 := #VAR.ENE_MWA3;
   #VAR_IF_ABP.EXT_HW := #VAR.EXT_HW;
   #VAR_IF_ABP.STO := #STO;
END_REGION
END_FUNCTION_BLOCK

FUNCTION_BLOCK "TYPIC_C501_IF_BBI"   // FB5, FBD
TITLE = TYPIC_C501_IF_BBI: Brandblusinstallatie
{ S7_Optimized_Access := 'TRUE' }
AUTHOR : OCOTECH
FAMILY : Typical
NAME : C501.701
// Logisch Object Besturing: C501.701
// 
// De interne functie brandblusinstallatie verwerkt de algemene bedieningen vanop het aanraakscherm en de algemene sturingen van de brandblusinstallatie.
// stored: MemoryReserve 10, SetENOAutomatically false
   VAR_INPUT
      EXT_HW { ExternalAccessible := 'False'; ExternalVisible := 'False'; ExternalWritable := 'False'} : Bool;   // Sturings hardware (PLC) bewaking (1 = OK)
      IN_STS1 { ExternalAccessible := 'False'; ExternalVisible := 'False'; ExternalWritable := 'False'} : Bool;   // Status schuif ALSB ingeschakeld
      IN_STS2 { ExternalAccessible := 'False'; ExternalVisible := 'False'; ExternalWritable := 'False'} : Bool;   // Status schuif ALSB in test
      IN_STS3 { ExternalAccessible := 'False'; ExternalVisible := 'False'; ExternalWritable := 'False'} : Bool;   // Status schuif ALSB uitgereden
      IN_AUT { ExternalAccessible := 'False'; ExternalVisible := 'False'; ExternalWritable := 'False'} : Bool;   // Beveiliging in ALSB-bord (1 = OK)
      IN_NB_AUT { ExternalAccessible := 'False'; ExternalVisible := 'False'; ExternalWritable := 'False'} : Bool;   // Beveiliging No-Break (1 = OK)
      IN_SPD_OK { ExternalAccessible := 'False'; ExternalVisible := 'False'; ExternalWritable := 'False'} : Bool;   // Status overspanningsbeveiliging (1 = OK)
      IN_KST_AUT { ExternalAccessible := 'False'; ExternalVisible := 'False'; ExternalWritable := 'False'} : Bool;   // Beveiliging kastklimatisatie (1 = OK)
      IN_KST_AAN { ExternalAccessible := 'False'; ExternalVisible := 'False'; ExternalWritable := 'False'} : Bool;   // Lastscheider aan (1 = AAN)
      IN_LDE { ExternalAccessible := 'False'; ExternalVisible := 'False'; ExternalWritable := 'False'} : Bool;   // Lekdetectie in pomplokaal (1 = OK)
   END_VAR
   VAR_OUTPUT
      VAR_IF_BBI { ExternalAccessible := 'False'; ExternalVisible := 'False'; ExternalWritable := 'False'} : "C501_VAR_IF_BBI_TYPIC";   // Struct met alle variabelen naar de basisfunctie
   END_VAR
   VAR_IN_OUT
      STU_IF_BBI : "C501_STU_IF_BBI_TYPIC";   // Struct met alle sturingen vanuit de basisfunctie
   END_VAR
   VAR
      BED : Struct   // Bedieningen
         UIT : Bool;   // Bediening om regime Uit te activeren
         BWK : Bool;   // Bediening om regime Bewaken te activeren
         BLUS1 : Bool;   // Bediening om regime Blussen Hydrant te activeren
         BLUS2 : Bool;   // Bediening om regime Blussen Hydrant en WMS te activeren
         TEST : Bool;   // Bediening om regime Testen te activeren
      END_STRUCT;
      STO { ExternalWritable := 'False'} : Struct   // Storingen
         A001 : Bool;   // Beveiliging aangesproken
         A002 : Bool;   // Beveiliging No-Break aangesproken
         A003 : Bool;   // Schuif ALSB uitgeschakeld
         A004 : Bool;   // Schuif ALSB in test
         A005 : Bool;   // Schuif ALSB uitgereden
         A006 : Bool;   // Lekdetectie in pomplokaal
         A007 : Bool;   // Overspanningsbeveiliging aangesproken
         A008 : Bool;   // Beveiliging kastklimatisatie aangesproken
         A009 : Bool;   // Lastscheider niet aan
      END_STRUCT;
      VAR { ExternalWritable := 'False'} : Struct   // Variabelen
         WRE : USInt;   // Actueel actief regime
         REQ_UIT { ExternalAccessible := 'False'; ExternalVisible := 'False'} : Bool;   // Aanvraag om regime Uit te activeren
         REQ_BWK { ExternalAccessible := 'False'; ExternalVisible := 'False'} : Bool;   // Aanvraag om regime Bewaken te activeren
         REQ_BLUS1 { ExternalAccessible := 'False'; ExternalVisible := 'False'} : Bool;   // Aanvraag om regime Blussen Hydrant te activeren
         REQ_BLUS2 { ExternalAccessible := 'False'; ExternalVisible := 'False'} : Bool;   // Aanvraag om regime Blussen Hydrant en WMS te activeren
         REQ_TEST { ExternalAccessible := 'False'; ExternalVisible := 'False'} : Bool;   // Aanvraag om regime Testen te activeren
         EXT_HW { ExternalAccessible := 'False'; ExternalVisible := 'False'} : Bool;   // Sturings hardware (PLC) in storing
      END_STRUCT;
   END_VAR
BEGIN

REGION Network 1: START
END_REGION

REGION Network 2: +++ Bedieningen +++
   // Verwerking van de bedieningen.
END_REGION

REGION Network 3: +++ Storingen +++
   // Verwerken van de storingsmeldingen.
END_REGION

REGION Network 4: Storing A001: Beveiliging aangesproken
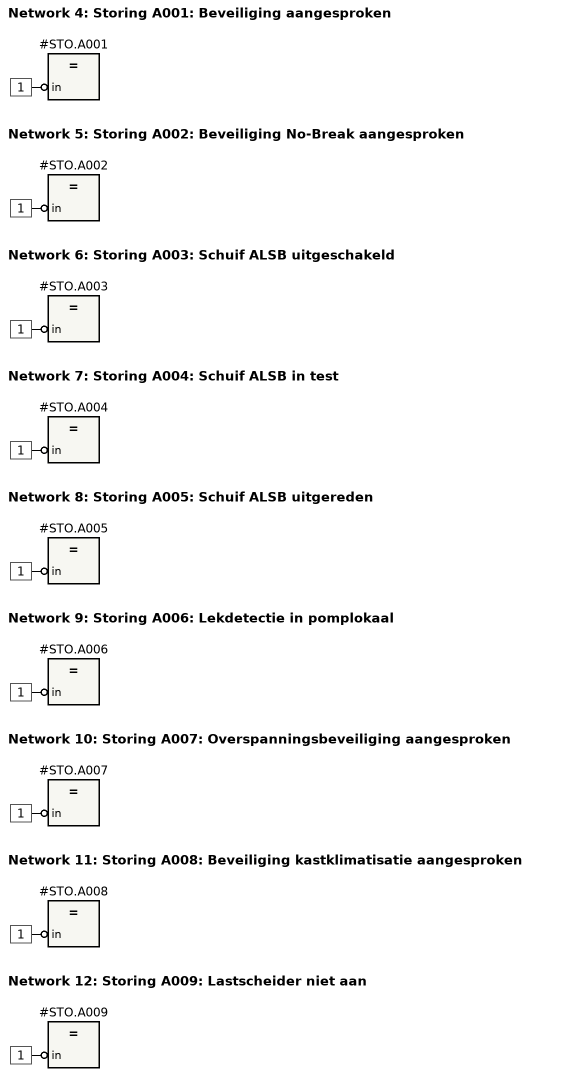
   #STO.A001 := NOT 1;
END_REGION

REGION Network 5: Storing A002: Beveiliging No-Break aangesproken
   #STO.A002 := NOT 1;
END_REGION

REGION Network 6: Storing A003: Schuif ALSB uitgeschakeld
   #STO.A003 := NOT 1;
END_REGION

REGION Network 7: Storing A004: Schuif ALSB in test
   #STO.A004 := NOT 1;
END_REGION

REGION Network 8: Storing A005: Schuif ALSB uitgereden
   #STO.A005 := NOT 1;
END_REGION

REGION Network 9: Storing A006: Lekdetectie in pomplokaal
   #STO.A006 := NOT 1;
END_REGION

REGION Network 10: Storing A007: Overspanningsbeveiliging aangesproken
   #STO.A007 := NOT 1;
END_REGION

REGION Network 11: Storing A008: Beveiliging kastklimatisatie aangesproken
   #STO.A008 := NOT 1;
END_REGION

REGION Network 12: Storing A009: Lastscheider niet aan
   #STO.A009 := NOT 1;
END_REGION

REGION Network 13: +++ Actieve werkingsregime aangeven +++
   // Het actieve werkingsregime wordt ontvangen vanuit de basisfunctie en wordt naar een interne variabele weggeschreven zodat het actieve werkingsregime kan aangegeven worden op het aanraakscherm.
END_REGION

REGION Network 14 (SCL): EINDE
   // Variabelen van intern scada rakvlak naar outputs copieren
   #VAR_IF_BBI.REQ_UIT := #VAR.REQ_UIT;
   #VAR_IF_BBI.REQ_BWK := #VAR.REQ_BWK;
   #VAR_IF_BBI.REQ_BLUS1 := #VAR.REQ_BLUS1;
   #VAR_IF_BBI.REQ_BLUS2 := #VAR.REQ_BLUS2;
   #VAR_IF_BBI.REQ_TEST := #VAR.REQ_TEST;
   #VAR_IF_BBI.EXT_HW := #VAR.EXT_HW;
   #VAR_IF_BBI.STO := #STO;
END_REGION
END_FUNCTION_BLOCK

FUNCTION_BLOCK "TYPIC_C501_IF_BBP"   // FB19, FBD
TITLE = TYPIC_C501_IF_BBP: Brandbluspomp
{ S7_Optimized_Access := 'TRUE' }
AUTHOR : OCOTECH
FAMILY : Typical
NAME : C501.707
// Logisch Object Besturing: C501.707
// 
// De interne functie brandbluspomp verzorgt de interne besturing, bewaking en fysieke aansturing van een brandbluspomp behorend tot de brandblusinstallatie.
// stored: MemoryReserve 10, SetENOAutomatically false
   VAR_INPUT
      PULS_100ms { ExternalAccessible := 'False'; ExternalVisible := 'False'; ExternalWritable := 'False'} : Bool;   // Puls, 1 PLC-cyclus hoog, 1 keer per 100 ms
      PULS_1s { ExternalAccessible := 'False'; ExternalVisible := 'False'; ExternalWritable := 'False'} : Bool;   // Puls, 1 PLC-cyclus hoog, 1 keer per seconde
      EXT_HW { ExternalAccessible := 'False'; ExternalVisible := 'False'; ExternalWritable := 'False'} : Bool;   // Sturings hardware (PLC) bewaking (1 = OK)
      IN_HND { ExternalAccessible := 'False'; ExternalVisible := 'False'; ExternalWritable := 'False'} : Bool;   // Terugmelding aansturing via hand (hardware)
      IN_AAN { ExternalAccessible := 'False'; ExternalVisible := 'False'; ExternalWritable := 'False'} : Bool;   // Terugmelding aansturing
      IN_AUT_C501 { ExternalAccessible := 'False'; ExternalVisible := 'False'; ExternalWritable := 'False'} : Bool;   // Beveiligingen: serie geschakelde terugmelding (1= OK)
      IN_AUT { ExternalAccessible := 'False'; ExternalVisible := 'False'; ExternalWritable := 'False'} : Bool;   // Status thermische beveiliging (1 = OK)
      IN_PTC { ExternalAccessible := 'False'; ExternalVisible := 'False'; ExternalWritable := 'False'} : Bool;   // Detectie hoge temperatuur in de wikkelingen van de motor (1 = OK)
      IN_SCW { ExternalAccessible := 'False'; ExternalVisible := 'False'; ExternalWritable := 'False'} : Bool;   // Werkschakelaar (1 = Aan)
      IN_STO { ExternalAccessible := 'False'; ExternalVisible := 'False'; ExternalWritable := 'False'} : Bool;   // Status Softstarter (1 = OK)
      IN_DME_STO { ExternalAccessible := 'False'; ExternalVisible := 'False'; ExternalWritable := 'False'} : Bool;   // Filterbewaking (1= OK / 0 = Vervuild)
      IN_STS1 { ExternalAccessible := 'False'; ExternalVisible := 'False'; ExternalWritable := 'False'} : Bool;   // Status motorlade ingeschakeld
      IN_STS2 { ExternalAccessible := 'False'; ExternalVisible := 'False'; ExternalWritable := 'False'} : Bool;   // Status motorlade in test
      IN_STS3 { ExternalAccessible := 'False'; ExternalVisible := 'False'; ExternalWritable := 'False'} : Bool;   // Status motorlade uitgereden
      IN_STR1 { ExternalAccessible := 'False'; ExternalVisible := 'False'; ExternalWritable := 'False'} : Int;   // Analoge meting ventilator fasestroom 1
      IN_STR2 { ExternalAccessible := 'False'; ExternalVisible := 'False'; ExternalWritable := 'False'} : Int;   // Analoge meting ventilator fasestroom 2
      IN_STR3 { ExternalAccessible := 'False'; ExternalVisible := 'False'; ExternalWritable := 'False'} : Int;   // Analoge meting ventilator fasestroom 3
      IN_TRL { ExternalAccessible := 'False'; ExternalVisible := 'False'; ExternalWritable := 'False'} : Bool;   // Trillingsdetectie (1 = Geen trillingen)
      CFG_TYD_FB { ExternalAccessible := 'False'; ExternalVisible := 'False'; ExternalWritable := 'False'} : Time;   // Vertragingstijd storing foute terugmelding
      CFG_TYD_TRL { ExternalAccessible := 'False'; ExternalVisible := 'False'; ExternalWritable := 'False'} : Time;   // Vertragingstijd storing onbalans
      CFG_TRL_MAX { ExternalAccessible := 'False'; ExternalVisible := 'False'; ExternalWritable := 'False'} : Real;   // Hoogste waarde scalering trillingsmeting
      CFG_TRL_MIN { ExternalAccessible := 'False'; ExternalVisible := 'False'; ExternalWritable := 'False'} : Real;   // Laagste waarde scalering trillingsmeting
      CFG_TRL_HOOG { ExternalAccessible := 'False'; ExternalVisible := 'False'; ExternalWritable := 'False'} : Real;   // Schakeldrempel hoog trillingsmeting (onbalans)
      CFG_TYD_RUN { ExternalAccessible := 'False'; ExternalVisible := 'False'; ExternalWritable := 'False'} : LInt;   // Minimale draaitijd om melding onderhoud nodig te resetten
      CFG_TYD_STOP { ExternalAccessible := 'False'; ExternalVisible := 'False'; ExternalWritable := 'False'} : LInt;   // Stilstandstijd die melding onderhoud nodig activeert
      CFG_TYD_MAX { ExternalAccessible := 'False'; ExternalVisible := 'False'; ExternalWritable := 'False'} : Int;   // Tijdsduur draaitijd overschrijding pomp
   END_VAR
   VAR_OUTPUT
      VAR_IF_BBP { ExternalAccessible := 'False'; ExternalVisible := 'False'; ExternalWritable := 'False'} : "C501_VAR_IF_BBP_TYPIC";   // Struct met alle variabelen naar bovenliggende functies
      OUT_AAN { ExternalAccessible := 'False'; ExternalVisible := 'False'; ExternalWritable := 'False'} : Bool;   // Aansturen pomp
      OUT_RES { ExternalAccessible := 'False'; ExternalVisible := 'False'; ExternalWritable := 'False'} : Bool;   // Reset softstarter
   END_VAR
   VAR_IN_OUT
      STU_IF_BBP : "C501_STU_IF_BBP_TYPIC";   // Struct met alle sturingen van de subfunctie (SF) pomp van 3B
   END_VAR
   VAR
      BED : Struct   // Bedieningen
         REM : Bool;   // Bediening om pomp in Remote te schakelen (indien IN_HND = 0)
         FWD : Bool;   // Bediening om pomp in hand te schakelen en te starten
         STOP : Bool;   // Bediening om pomp in hand te schakelen en te stoppen
         RES : Bool;   // Reset storingen
      END_STRUCT;
      STO { ExternalWritable := 'False'} : Struct   // Storingen
         A001 : Bool;   // Beveiliging aangesproken
         A002 : Bool;   // Storing van de motorbeveiliging van de pomp
         A003 : Bool;   // Storing softstarter
         A004 : Bool;   // Te hoge temperatuur in de motorwikkelingen
         A005 : Bool;   // De pomp is in onbalans
         A006 : Bool;   // Motorlade uitgeschakeld
         A007 : Bool;   // Motorlade in test
         A008 : Bool;   // Motorlade uitgereden
         A009 : Bool;   // Fout stroommeting fase 1
         A010 : Bool;   // Fout stroommeting fase 2
         A011 : Bool;   // Fout stroommeting fase 3
         A012 : Bool;   // Filter vervuild
         AT01 : Bool;   // Discordantie motor: terugmelding niet ontvangen
         AT02 : Bool;   // Discordantie motor: terugmelding blijft aanwezig
         M001 : Bool;   // Werkschakelaar uitgeschakeld
         M002 : Bool;   // Melding: Pomp heeft te lang niet gedraaid. Periodiek onderhoud nodig
         M003 : Bool;   // Melding: Draaitijd overschrijding
      END_STRUCT;
      VAR { ExternalWritable := 'False'} : Struct   // Variabelen
         STS_AAN : Bool;   // Pomp draait
         BMO_HAND : Bool;   // Pomp in hand geschakeld
         TYD_TOT_AAN { ExternalAccessible := 'False'; ExternalVisible := 'False'} : LInt;   // Totaal aantal draaiuren (in seconden)
         TYD_TOT_AAN_UUR { ExternalAccessible := 'False'; ExternalVisible := 'False'} : LInt;   // Totaal aantal draaiuren (in uren)
         TYD_AAN { ExternalAccessible := 'False'; ExternalVisible := 'False'} : Int;   // Aantal seconden dat pomp aangeschakeld is
         TYD_UIT { ExternalAccessible := 'False'; ExternalVisible := 'False'} : Int;   // Aantal seconden dat pomp uitgeschakeld is
         ENE_MWA1 { ExternalAccessible := 'False'; ExternalVisible := 'False'} : Real;   // Stroommeting fase 1
         ENE_MWA2 { ExternalAccessible := 'False'; ExternalVisible := 'False'} : Real;   // Stroommeting fase 2
         ENE_MWA3 { ExternalAccessible := 'False'; ExternalVisible := 'False'} : Real;   // Stroommeting fase 3
         EXT_HW { ExternalAccessible := 'False'; ExternalVisible := 'False'} : Bool;   // Sturings hardware (PLC) in storing
      END_STRUCT;
   END_VAR
BEGIN

REGION Network 1: START
END_REGION

REGION Network 2: +++ Metingen +++
   // Inlezen van de 3 stroommetingen van iedere fase van de motor.
END_REGION

REGION Network 3: +++ Storingen +++
   // Verwerken van de storingsmeldingen (inputs).
END_REGION

REGION Network 4: Storing A001: Beveiliging aangesproken
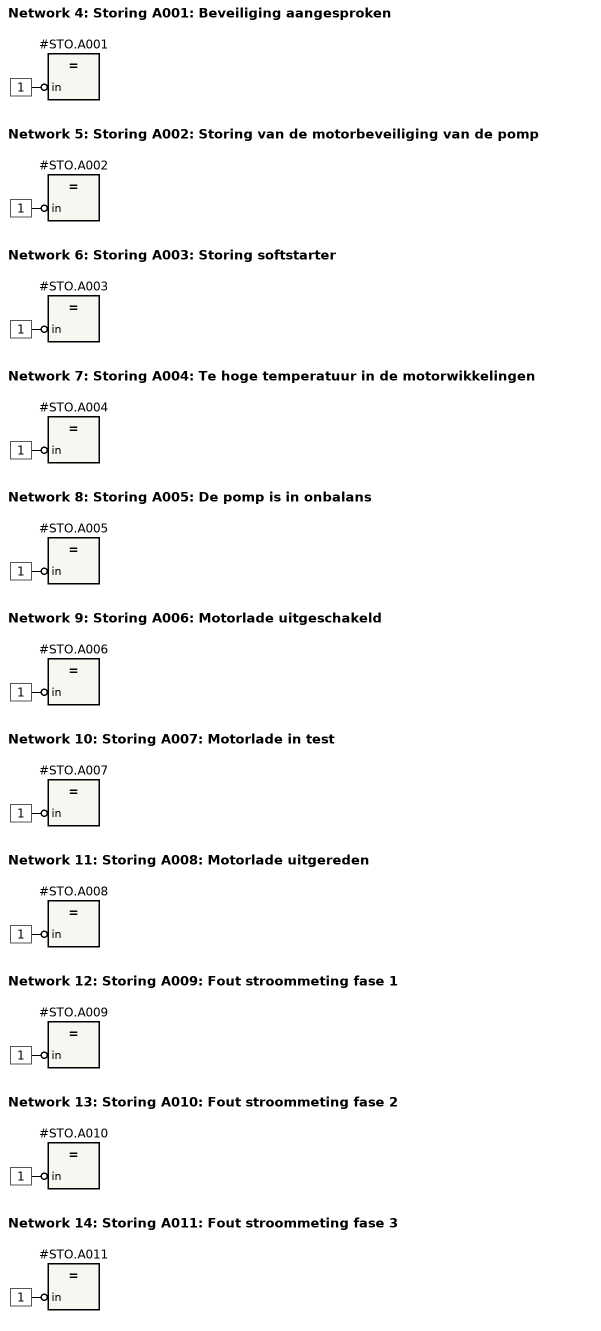
   #STO.A001 := NOT 1;
END_REGION

REGION Network 5: Storing A002: Storing van de motorbeveiliging van de pomp
   #STO.A002 := NOT 1;
END_REGION

REGION Network 6: Storing A003: Storing softstarter
   #STO.A003 := NOT 1;
END_REGION

REGION Network 7: Storing A004: Te hoge temperatuur in de motorwikkelingen
   #STO.A004 := NOT 1;
END_REGION

REGION Network 8: Storing A005: De pomp is in onbalans
   #STO.A005 := NOT 1;
END_REGION

REGION Network 9: Storing A006: Motorlade uitgeschakeld
   #STO.A006 := NOT 1;
END_REGION

REGION Network 10: Storing A007: Motorlade in test
   #STO.A007 := NOT 1;
END_REGION

REGION Network 11: Storing A008: Motorlade uitgereden
   #STO.A008 := NOT 1;
END_REGION

REGION Network 12: Storing A009: Fout stroommeting fase 1
   #STO.A009 := NOT 1;
END_REGION

REGION Network 13: Storing A010: Fout stroommeting fase 2
   #STO.A010 := NOT 1;
END_REGION

REGION Network 14: Storing A011: Fout stroommeting fase 3
   #STO.A011 := NOT 1;
END_REGION

REGION Network 15: Storing A012: Filter vervuild
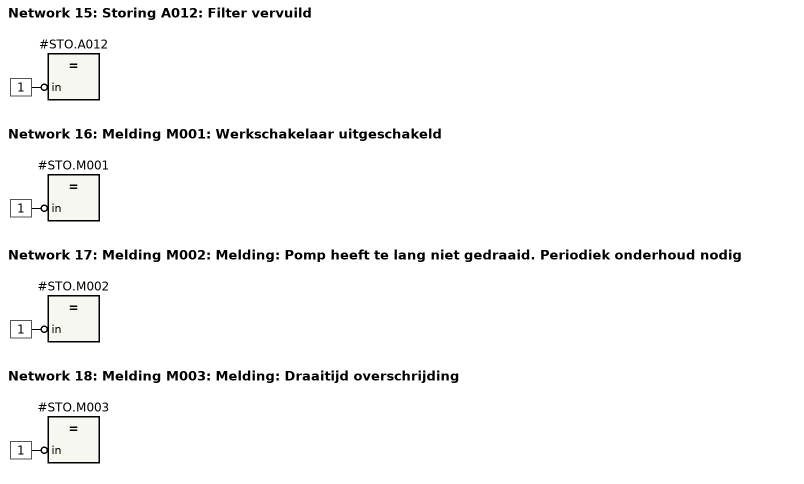
   #STO.A012 := NOT 1;
END_REGION

REGION Network 16: Melding M001: Werkschakelaar uitgeschakeld
   #STO.M001 := NOT 1;
END_REGION

REGION Network 17: Melding M002: Melding: Pomp heeft te lang niet gedraaid. Periodiek onderhoud nodig
   #STO.M002 := NOT 1;
END_REGION

REGION Network 18: Melding M003: Melding: Draaitijd overschrijding
   #STO.M003 := NOT 1;
END_REGION

REGION Network 19: +++ Motorsturing +++
   // Aansturen en bewaking van de motor.
END_REGION

REGION Network 20: +++ Urentellers +++
   // Tellen van de tijdsduur dat motor draait of stilstaat.
END_REGION

REGION Network 21 (SCL): EINDE
   // Variabelen van intern scada rakvlak naar outputs copieren
   #VAR_IF_BBP.STS_AAN := #VAR.STS_AAN;
   #VAR_IF_BBP.BMO_HAND := #VAR.BMO_HAND;
   #VAR_IF_BBP.TYD_TOT_AAN := #VAR.TYD_TOT_AAN;
   #VAR_IF_BBP.TYD_TOT_AAN_UUR := #VAR.TYD_TOT_AAN_UUR;
   #VAR_IF_BBP.TYD_AAN := #VAR.TYD_AAN;
   #VAR_IF_BBP.TYD_UIT := #VAR.TYD_UIT;
   #VAR_IF_BBP.ENE_MWA1 := #VAR.ENE_MWA1;
   #VAR_IF_BBP.ENE_MWA2 := #VAR.ENE_MWA2;
   #VAR_IF_BBP.ENE_MWA3 := #VAR.ENE_MWA3;
   #VAR_IF_BBP.EXT_HW := #VAR.EXT_HW;
   #VAR_IF_BBP.STO := #STO;
END_REGION
END_FUNCTION_BLOCK

FUNCTION_BLOCK "TYPIC_C501_IF_DME"   // FB34, FBD
TITLE = TYPIC_C501_IF_DME: Drukmeting
{ S7_Optimized_Access := 'TRUE' }
AUTHOR : OCOTECH
FAMILY : Typical
NAME : C501.710
// Logisch Object Besturing: C501.710
// 
// De interne functie drukmeting verzorgt de interne besturing en bewaking van een drukmeting.
// stored: MemoryReserve 10, SetENOAutomatically false
   VAR_INPUT
      EXT_HW { ExternalAccessible := 'False'; ExternalVisible := 'False'; ExternalWritable := 'False'} : Bool;   // Sturings hardware (PLC) bewaking (1 = OK)
      IN_MWA { ExternalAccessible := 'False'; ExternalVisible := 'False'; ExternalWritable := 'False'} : Word;   // Meetwaarde
      IN_AUT_C501 { ExternalAccessible := 'False'; ExternalVisible := 'False'; ExternalWritable := 'False'} : Bool;   // Beveiligingen: serie geschakelde terugmelding (1= OK)
      CFG_MAX_SWA { ExternalAccessible := 'False'; ExternalVisible := 'False'; ExternalWritable := 'False'} : Real;   // Maximale waarde temperatuurmeting
      CFG_MIN_SWA { ExternalAccessible := 'False'; ExternalVisible := 'False'; ExternalWritable := 'False'} : Real;   // Minimale waarde temperatuurmeting
   END_VAR
   VAR_OUTPUT
      VAR_IF_DME { ExternalAccessible := 'False'; ExternalVisible := 'False'; ExternalWritable := 'False'} : "C501_VAR_IF_DME_TYPIC";   // Struct met alle variabelen naar bovenliggende functies
   END_VAR
   VAR
      STO { ExternalWritable := 'False'} : Struct   // Storingen
         A001 : Bool;   // Beveiliging aangesproken
         A002 : Bool;   // Draadbreuk analoge meting
         A003 : Bool;   // Meetbereik overschreden
         A004 : Bool;   // Drukmeter geeft storing
      END_STRUCT;
      VAR { ExternalWritable := 'False'} : Struct   // Variabelen
         MWA : Real;   // Meetwaarde
         EXT_HW { ExternalAccessible := 'False'; ExternalVisible := 'False'} : Bool;   // Sturings hardware (PLC) in storing
      END_STRUCT;
   END_VAR
BEGIN

REGION Network 1: START
END_REGION

REGION Network 2: +++ Verwerking analoge meting +++
   // Verwerking analoge meting naar een meetwaarde in m3/u en detectie storingen van de meting.
END_REGION

REGION Network 3: +++ Storingen +++
   // Storingen van de analoge meting.
END_REGION

REGION Network 4: Storing A001: Beveiliging aangesproken
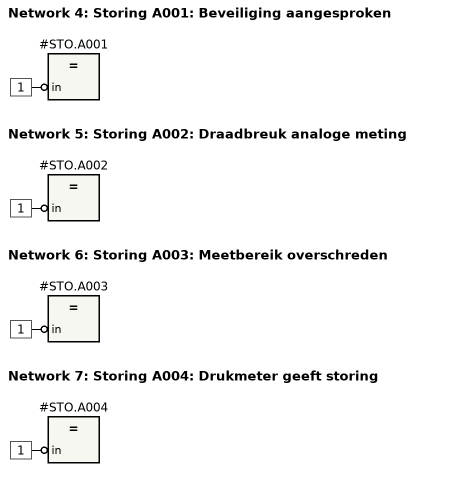
   #STO.A001 := NOT 1;
END_REGION

REGION Network 5: Storing A002: Draadbreuk analoge meting
   #STO.A002 := NOT 1;
END_REGION

REGION Network 6: Storing A003: Meetbereik overschreden
   #STO.A003 := NOT 1;
END_REGION

REGION Network 7: Storing A004: Drukmeter geeft storing
   #STO.A004 := NOT 1;
END_REGION

REGION Network 8 (SCL): EINDE
   // Variabelen van intern scada rakvlak naar outputs copieren
   #VAR_IF_DME.MWA := #VAR.MWA;
   #VAR_IF_DME.EXT_HW := #VAR.EXT_HW;
   #VAR_IF_DME.STO := #STO;
END_REGION
END_FUNCTION_BLOCK

FUNCTION_BLOCK "TYPIC_C501_IF_HYK"   // FB65, FBD
TITLE = TYPIC_C501_IF_HYK: Hydrantkast tunnelmond
{ S7_Optimized_Access := 'TRUE' }
AUTHOR : OCOTECH
FAMILY : Typical
NAME : C501.709
// Logisch Object Besturing: C501.709
// 
// De interne functie hydrantkast verzorgt de interne bewaking van een hydrantkast.
// stored: MemoryReserve 10, SetENOAutomatically false
   VAR_INPUT
      EXT_HW { ExternalAccessible := 'False'; ExternalVisible := 'False'; ExternalWritable := 'False'} : Bool;   // Sturings hardware (PLC) bewaking (1 = OK)
      IN_DEC { ExternalAccessible := 'False'; ExternalVisible := 'False'; ExternalWritable := 'False'} : Bool;   // De hydrantkast in de verkeerskoker is gesloten. (TRUE = Gesloten)
      IN_STO { ExternalAccessible := 'False'; ExternalVisible := 'False'; ExternalWritable := 'False'} : Bool;   // Temperatuursensor (TRUE = OK / FALSE = Storing)
      IN_AUT_C501 { ExternalAccessible := 'False'; ExternalVisible := 'False'; ExternalWritable := 'False'} : Bool;   // Beveiligingen: serie geschakelde terugmelding (1= OK)
   END_VAR
   VAR_OUTPUT
      VAR_IF_HYK { ExternalAccessible := 'False'; ExternalVisible := 'False'; ExternalWritable := 'False'} : "C501_VAR_IF_HYK_TYPIC";   // Struct met alle variabelen naar bovenliggende functies
   END_VAR
   VAR
      STO { ExternalWritable := 'False'} : Struct   // Storingen
         A001 : Bool;   // Beveiliging aangesproken
         A002 : Bool;   // Temperatuur te laag
      END_STRUCT;
      VAR { ExternalWritable := 'False'} : Struct   // Variabelen
         DEC : Bool;   // De hydrantkast in de verkeerskoker is gesloten
         EXT_HW { ExternalAccessible := 'False'; ExternalVisible := 'False'} : Bool;   // Sturings hardware (PLC) in storing
      END_STRUCT;
   END_VAR
BEGIN

REGION Network 1: START
END_REGION

REGION Network 2: +++ Storingen +++
   // Storingen van de hydrantkast.
END_REGION

REGION Network 3: Storing A001: Beveiliging aangesproken
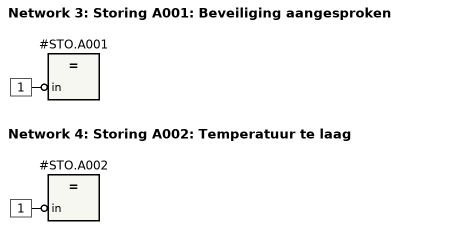
   #STO.A001 := NOT 1;
END_REGION

REGION Network 4: Storing A002: Temperatuur te laag
   #STO.A002 := NOT 1;
END_REGION

REGION Network 5: +++ Variabelen +++
   // Toestandsvariabelen naar 3B sturen
END_REGION

REGION Network 6 (SCL): EINDE
   // Variabelen van intern scada rakvlak naar outputs copieren
   #VAR_IF_HYK.DEC := #VAR.DEC;
   #VAR_IF_HYK.EXT_HW := #VAR.EXT_HW;
   #VAR_IF_HYK.STO := #STO;
END_REGION
END_FUNCTION_BLOCK

FUNCTION_BLOCK "TYPIC_C501_IF_JKP"   // FB35, FBD
TITLE = TYPIC_C501_IF_JKP: Jockeypomp
{ S7_Optimized_Access := 'TRUE' }
AUTHOR : OCOTECH
FAMILY : Typical
NAME : C501.706
// Logisch Object Besturing: C501.706
// 
// De interne functie pomp verzorgt de interne besturing, bewaking en fysieke aansturing van een jockeypomp behorend tot de brandblusinstallatie.
// stored: MemoryReserve 10, SetENOAutomatically false
   VAR_INPUT
      PULS_100ms { ExternalAccessible := 'False'; ExternalVisible := 'False'; ExternalWritable := 'False'} : Bool;   // Puls, 1 PLC-cyclus hoog, 1 keer per 100 ms
      PULS_1s { ExternalAccessible := 'False'; ExternalVisible := 'False'; ExternalWritable := 'False'} : Bool;   // Puls, 1 PLC-cyclus hoog, 1 keer per seconde
      EXT_HW { ExternalAccessible := 'False'; ExternalVisible := 'False'; ExternalWritable := 'False'} : Bool;   // Sturings hardware (PLC) bewaking (1 = OK)
      IN_AAN { ExternalAccessible := 'False'; ExternalVisible := 'False'; ExternalWritable := 'False'} : Bool;   // Terugmelding aansturing
      IN_AUT_C501 { ExternalAccessible := 'False'; ExternalVisible := 'False'; ExternalWritable := 'False'} : Bool;   // Beveiligingen: serie geschakelde terugmelding (1= OK)
      IN_AUT { ExternalAccessible := 'False'; ExternalVisible := 'False'; ExternalWritable := 'False'} : Bool;   // Status thermische beveiliging (1 = OK)
      IN_SCW { ExternalAccessible := 'False'; ExternalVisible := 'False'; ExternalWritable := 'False'} : Bool;   // Werkschakelaar (1 = Aan)
      IN_DME_STO { ExternalAccessible := 'False'; ExternalVisible := 'False'; ExternalWritable := 'False'} : Bool;   // Filterbewaking storing (0 = Storing)
      CFG_TYD_FB { ExternalAccessible := 'False'; ExternalVisible := 'False'; ExternalWritable := 'False'} : Time;   // Vertragingstijd storing foute terugmelding
   END_VAR
   VAR_OUTPUT
      VAR_IF_JKP { ExternalAccessible := 'False'; ExternalVisible := 'False'; ExternalWritable := 'False'} : "C501_VAR_IF_JKP_TYPIC";   // Struct met alle variabelen naar bovenliggende functies
      OUT_AAN { ExternalAccessible := 'False'; ExternalVisible := 'False'; ExternalWritable := 'False'} : Bool;   // Aansturen pomp
   END_VAR
   VAR_IN_OUT
      STU_IF_JKP : "C501_STU_IF_JKP_TYPIC";   // Struct met alle sturingen van de subfunctie (SF) jockeypomp van 3B
   END_VAR
   VAR
      BED : Struct   // Bedieningen
         REM : Bool;   // Bediening om pomp in Remote te schakelen (indien IN_HND = 0)
         FWD : Bool;   // Bediening om pomp in hand te schakelen en te starten
         STOP : Bool;   // Bediening om pomp in hand te schakelen en te stoppen
         RES : Bool;   // Reset storingen
      END_STRUCT;
      STO { ExternalWritable := 'False'} : Struct   // Storingen
         A001 : Bool;   // Beveiliging aangesproken
         A002 : Bool;   // Filter vervuild
         A003 : Bool;   // Storing van de motorbeveiliging van de pomp
         AT01 : Bool;   // Discordantie motor: terugmelding niet ontvangen
         AT02 : Bool;   // Discordantie motor: terugmelding blijft aanwezig
         M001 : Bool;   // Werkschakelaar uitgeschakeld
         M002 : Bool;   // Melding: Pomp heeft te lang niet gedraaid. Periodiek onderhoud nodig
      END_STRUCT;
      VAR { ExternalWritable := 'False'} : Struct   // Variabelen
         STS_AAN : Bool;   // Pomp draait
         BMO_HAND : Bool;   // Pomp in hand geschakeld
         TYD_TOT_AAN { ExternalAccessible := 'False'; ExternalVisible := 'False'} : LInt;   // Totaal aantal draaiuren in seconden
         TYD_TOT_AAN_UUR { ExternalAccessible := 'False'; ExternalVisible := 'False'} : LInt;   // Totaal aantal draaiuren (in uren)
         TYD_AAN { ExternalAccessible := 'False'; ExternalVisible := 'False'} : Int;   // Aantal seconden dat pomp aangeschakeld is
         TYD_UIT { ExternalAccessible := 'False'; ExternalVisible := 'False'} : Int;   // Aantal seconden dat pomp uitgeschakeld is
         EXT_HW { ExternalAccessible := 'False'; ExternalVisible := 'False'} : Bool;   // Sturings hardware (PLC) in storing
      END_STRUCT;
   END_VAR
BEGIN

REGION Network 1: START
END_REGION

REGION Network 2: +++ Storingen +++
   // Verwerken van de storingsmeldingen (inputs).
END_REGION

REGION Network 3: Storing A001: Beveiliging aangesproken
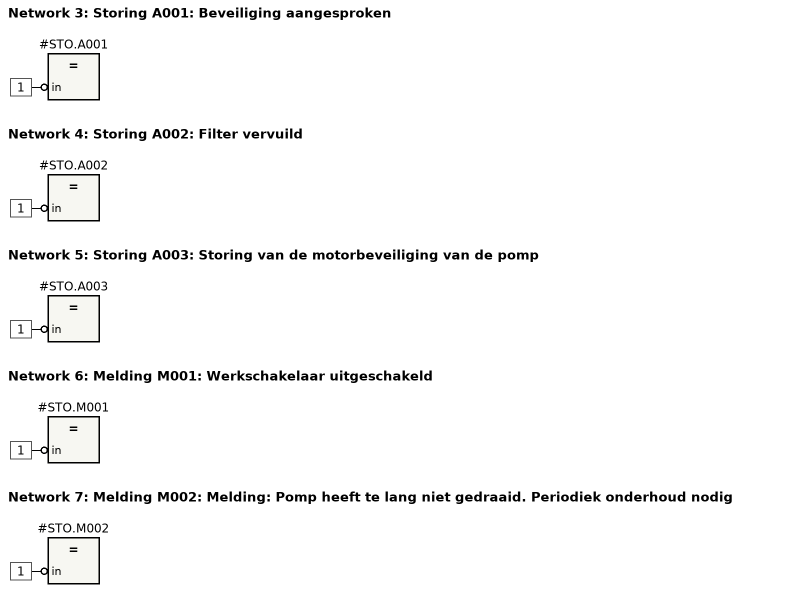
   #STO.A001 := NOT 1;
END_REGION

REGION Network 4: Storing A002: Filter vervuild
   #STO.A002 := NOT 1;
END_REGION

REGION Network 5: Storing A003: Storing van de motorbeveiliging van de pomp
   #STO.A003 := NOT 1;
END_REGION

REGION Network 6: Melding M001: Werkschakelaar uitgeschakeld
   #STO.M001 := NOT 1;
END_REGION

REGION Network 7: Melding M002: Melding: Pomp heeft te lang niet gedraaid. Periodiek onderhoud nodig
   #STO.M002 := NOT 1;
END_REGION

REGION Network 8: +++ Motorsturing +++
   // Aansturen en bewaking van de motor.
END_REGION

REGION Network 9: +++ Urentellers +++
   // Tellen van de tijdsduur dat motor draait of stilstaat.
END_REGION

REGION Network 10 (SCL): EINDE
   // Variabelen van intern scada rakvlak naar outputs copieren
   #VAR_IF_JKP.STS_AAN := #VAR.STS_AAN;
   #VAR_IF_JKP.BMO_HAND := #VAR.BMO_HAND;
   #VAR_IF_JKP.TYD_TOT_AAN := #VAR.TYD_TOT_AAN;
   #VAR_IF_JKP.TYD_TOT_AAN_UUR := #VAR.TYD_TOT_AAN_UUR;
   #VAR_IF_JKP.TYD_AAN := #VAR.TYD_AAN;
   #VAR_IF_JKP.TYD_UIT := #VAR.TYD_UIT;
   #VAR_IF_JKP.EXT_HW := #VAR.EXT_HW;
   #VAR_IF_JKP.STO := #STO;
END_REGION
END_FUNCTION_BLOCK

FUNCTION_BLOCK "TYPIC_C501_IF_KLG"   // FB64, FBD
TITLE = TYPIC_C501_IF_KLG: Motorgestuurde klep
{ S7_Optimized_Access := 'TRUE' }
AUTHOR : OCOTECH
FAMILY : Typical
NAME : C501.703
// Logisch Object Besturing: C501.703
// 
// De interne functie motorgestuurde klep verzorgt de interne besturing, bewaking en fysieke aansturing van een motorgestuurde klep behorend tot de brandblusinstallatie.
// stored: MemoryReserve 10, SetENOAutomatically false
   VAR_INPUT
      EXT_HW { ExternalAccessible := 'False'; ExternalVisible := 'False'; ExternalWritable := 'False'} : Bool;   // Sturings hardware (PLC) bewaking (1 = OK)
      IN_OPEN { ExternalAccessible := 'False'; ExternalVisible := 'False'; ExternalWritable := 'False'} : Bool;   // Klep is open
      IN_TOE { ExternalAccessible := 'False'; ExternalVisible := 'False'; ExternalWritable := 'False'} : Bool;   // Klep is toe
      IN_AUT_C501 { ExternalAccessible := 'False'; ExternalVisible := 'False'; ExternalWritable := 'False'} : Bool;   // Beveiligingen: serie geschakelde terugmelding (1= OK)
      CFG_TYD_FB { ExternalAccessible := 'False'; ExternalVisible := 'False'; ExternalWritable := 'False'} : Time;   // Vertragingstijd storing foute terugmelding
   END_VAR
   VAR_OUTPUT
      VAR_IF_KLG { ExternalAccessible := 'False'; ExternalVisible := 'False'; ExternalWritable := 'False'} : "C501_VAR_IF_KLG_TYPIC";   // Struct met alle variabelen naar bovenliggende functies
      OUT_OPEN { ExternalAccessible := 'False'; ExternalVisible := 'False'; ExternalWritable := 'False'} : Bool;   // Klep openen
      OUT_TOE { ExternalAccessible := 'False'; ExternalVisible := 'False'; ExternalWritable := 'False'} : Bool;   // Klep sluiten
   END_VAR
   VAR_IN_OUT
      STU_IF_KLG : "C501_STU_IF_KLG_TYPIC";   // Struct met alle sturingen van de subfunctie (SF) motorgestuurde klep van 3B
   END_VAR
   VAR
      BED : Struct   // Bedieningen
         REM : Bool;   // Bediening om klep in Remote te schakelen (indien IN_HND = 0)
         OPEN : Bool;   // Bediening om klep in hand te schakelen en te openen
         TOE : Bool;   // Bediening om klep in hand te schakelen en te sluiten
         RES : Bool;   // Reset storingen
      END_STRUCT;
      STO { ExternalWritable := 'False'} : Struct   // Storingen
         A001 : Bool;   // Beveiliging aangesproken
         AT01 : Bool;   // Terugmelding Open niet ontvangen
         AT02 : Bool;   // Terugmelding Dicht niet ontvangen
         AT03 : Bool;   // Terugmeldingen Open en Dicht tegelijkertijd
      END_STRUCT;
      VAR { ExternalWritable := 'False'} : Struct   // Variabelen
         HAND_OPEN { ExternalAccessible := 'False'; ExternalVisible := 'False'} : Bool;   // TRUE = Gewenste stand in hand is Open FALSE = Gewenste stand in hand is Toe
         CMD_OPEN { ExternalAccessible := 'False'; ExternalVisible := 'False'} : Bool;   // TRUE = Gewenste stand is Open FALSE = Gewenste stand is Toe
         STS_OPEN : Bool;   // Motorgestuurde klep is open
         STS_TOE : Bool;   // Motorgestuurde klep is toe
         STS_BEZ_OPEN : Bool;   // Motorgestuurde klep is aan het openen (1 = Open)
         STS_BEZ_TOE : Bool;   // Motorgestuurde klep is aan het sluiten (1 = Toe)
         BMO_HAND : Bool;   // TRUE = in hand geschakeld FALSE = niet in hand
         EXT_HW { ExternalAccessible := 'False'; ExternalVisible := 'False'} : Bool;   // Sturings hardware (PLC) in storing
      END_STRUCT;
   END_VAR
BEGIN

REGION Network 1: START
END_REGION

